	LOCAL CONST Robtarget Tr_meulage_motif_1_P373 :=[[-210.10528125,-32.02706640625,-17.9608046875],[0.732123189175605,-0.57971865199821,0.222030212103854,-0.280400615744397],[0,0,0,0],[8.999999E+09,8.999999E+09,8.999999E+09,8.999999E+09,8.999999E+09,8.999999E+09]];
	LOCAL CONST Robtarget Tr_meulage_motif_1_P374 :=[[-209.3355625,-32.6537734375,-18.0711484375],[0.732123189175605,-0.57971865199821,0.222030212103854,-0.280400615744397],[0,0,0,0],[8.999999E+09,8.999999E+09,8.999999E+09,8.999999E+09,8.999999E+09,8.999999E+09]];
	LOCAL CONST Robtarget Tr_meulage_motif_1_P375 :=[[-208.563984375,-33.28990625,-18.07105078125],[0.732123189175605,-0.57971865199821,0.222030212103854,-0.280400615744397],[0,0,0,0],[8.999999E+09,8.999999E+09,8.999999E+09,8.999999E+09,8.999999E+09,8.999999E+09]];
	LOCAL CONST Robtarget Tr_meulage_motif_1_P376 :=[[-207.79240625,-33.9260390625,-18.070953125],[0.732123189175605,-0.57971865199821,0.222030212103854,-0.280400615744397],[0,0,0,0],[8.999999E+09,8.999999E+09,8.999999E+09,8.999999E+09,8.999999E+09,8.999999E+09]];
	LOCAL CONST Robtarget Tr_meulage_motif_1_P377 :=[[-207.020828125,-34.56217578125,-18.070853515625],[0.732123189175605,-0.57971865199821,0.222030212103854,-0.280400615744397],[0,0,0,0],[8.999999E+09,8.999999E+09,8.999999E+09,8.999999E+09,8.999999E+09,8.999999E+09]];
	LOCAL CONST Robtarget Tr_meulage_motif_1_P378 :=[[-206.24925,-35.19830859375,-18.070755859375],[0.732123189175605,-0.57971865199821,0.222030212103854,-0.280400615744397],[0,0,0,0],[8.999999E+09,8.999999E+09,8.999999E+09,8.999999E+09,8.999999E+09,8.999999E+09]];
	LOCAL CONST Robtarget Tr_meulage_motif_1_P379 :=[[-205.47765625,-35.83444140625,-18.07065625],[0.732123189175605,-0.57971865199821,0.222030212103854,-0.280400615744397],[0,0,0,0],[8.999999E+09,8.999999E+09,8.999999E+09,8.999999E+09,8.999999E+09,8.999999E+09]];
	LOCAL CONST Robtarget Tr_meulage_motif_1_P380 :=[[-204.706078125,-36.47057421875,-18.07055859375],[0.732123189175605,-0.57971865199821,0.222030212103854,-0.280400615744397],[0,0,0,0],[8.999999E+09,8.999999E+09,8.999999E+09,8.999999E+09,8.999999E+09,8.999999E+09]];
	LOCAL CONST Robtarget Tr_meulage_motif_1_P381 :=[[-203.9345,-37.10670703125,-18.0704609375],[0.732123189175605,-0.57971865199821,0.222030212103854,-0.280400615744397],[0,0,0,0],[8.999999E+09,8.999999E+09,8.999999E+09,8.999999E+09,8.999999E+09,8.999999E+09]];
	LOCAL CONST Robtarget Tr_meulage_motif_1_P382 :=[[-203.162921875,-37.74283984375,-18.070361328125],[0.732123189175605,-0.57971865199821,0.222030212103854,-0.280400615744397],[0,0,0,0],[8.999999E+09,8.999999E+09,8.999999E+09,8.999999E+09,8.999999E+09,8.999999E+09]];
	LOCAL CONST Robtarget Tr_meulage_motif_1_P383 :=[[-202.39134375,-38.37897265625,-18.070263671875],[0.732123189175605,-0.57971865199821,0.222030212103854,-0.280400615744397],[0,0,0,0],[8.999999E+09,8.999999E+09,8.999999E+09,8.999999E+09,8.999999E+09,8.999999E+09]];
	LOCAL CONST Robtarget Tr_meulage_motif_1_P384 :=[[-201.619765625,-39.01510546875,-18.0701640625],[0.732123189175605,-0.57971865199821,0.222030212103854,-0.280400615744397],[0,0,0,0],[8.999999E+09,8.999999E+09,8.999999E+09,8.999999E+09,8.999999E+09,8.999999E+09]];
	LOCAL CONST Robtarget Tr_meulage_motif_1_P385 :=[[-200.8481875,-39.65123828125,-18.07006640625],[0.732123189175605,-0.57971865199821,0.222030212103854,-0.280400615744397],[0,0,0,0],[8.999999E+09,8.999999E+09,8.999999E+09,8.999999E+09,8.999999E+09,8.999999E+09]];
	LOCAL CONST Robtarget Tr_meulage_motif_1_P386 :=[[-200.076609375,-40.28737109375,-18.069966796875],[0.732123189175605,-0.57971865199821,0.222030212103854,-0.280400615744397],[0,0,0,0],[8.999999E+09,8.999999E+09,8.999999E+09,8.999999E+09,8.999999E+09,8.999999E+09]];
	LOCAL CONST Robtarget Tr_meulage_motif_1_P387 :=[[-199.30503125,-40.9235078125,-18.069869140625],[0.732123189175605,-0.57971865199821,0.222030212103854,-0.280400615744397],[0,0,0,0],[8.999999E+09,8.999999E+09,8.999999E+09,8.999999E+09,8.999999E+09,8.999999E+09]];
	LOCAL CONST Robtarget Tr_meulage_motif_1_P388 :=[[-198.533453125,-41.559640625,-18.069771484375],[0.732123189175605,-0.57971865199821,0.222030212103854,-0.280400615744397],[0,0,0,0],[8.999999E+09,8.999999E+09,8.999999E+09,8.999999E+09,8.999999E+09,8.999999E+09]];
	LOCAL CONST Robtarget Tr_meulage_motif_1_P389 :=[[-197.761875,-42.1957734375,-18.069671875],[0.732123189175605,-0.57971865199821,0.222030212103854,-0.280400615744397],[0,0,0,0],[8.999999E+09,8.999999E+09,8.999999E+09,8.999999E+09,8.999999E+09,8.999999E+09]];
	LOCAL CONST Robtarget Tr_meulage_motif_1_P390 :=[[-196.990296875,-42.83190625,-18.06957421875],[0.732123189175605,-0.57971865199821,0.222030212103854,-0.280400615744397],[0,0,0,0],[8.999999E+09,8.999999E+09,8.999999E+09,8.999999E+09,8.999999E+09,8.999999E+09]];
	LOCAL CONST Robtarget Tr_meulage_motif_1_P391 :=[[-196.21871875,-43.4680390625,-18.069474609375],[0.732123189175605,-0.57971865199821,0.222030212103854,-0.280400615744397],[0,0,0,0],[8.999999E+09,8.999999E+09,8.999999E+09,8.999999E+09,8.999999E+09,8.999999E+09]];
	LOCAL CONST Robtarget Tr_meulage_motif_1_P392 :=[[-195.447140625,-44.104171875,-18.069376953125],[0.732123189175605,-0.57971865199821,0.222030212103854,-0.280400615744397],[0,0,0,0],[8.999999E+09,8.999999E+09,8.999999E+09,8.999999E+09,8.999999E+09,8.999999E+09]];
	LOCAL CONST Robtarget Tr_meulage_motif_1_P393 :=[[-194.675546875,-44.7403046875,-18.069279296875],[0.732123189175605,-0.57971865199821,0.222030212103854,-0.280400615744397],[0,0,0,0],[8.999999E+09,8.999999E+09,8.999999E+09,8.999999E+09,8.999999E+09,8.999999E+09]];
	LOCAL CONST Robtarget Tr_meulage_motif_1_P394 :=[[-193.90396875,-45.3764375,-18.0691796875],[0.732123189175605,-0.57971865199821,0.222030212103854,-0.280400615744397],[0,0,0,0],[8.999999E+09,8.999999E+09,8.999999E+09,8.999999E+09,8.999999E+09,8.999999E+09]];
	LOCAL CONST Robtarget Tr_meulage_motif_1_P395 :=[[-193.132390625,-46.0125703125,-18.06908203125],[0.732123189175605,-0.57971865199821,0.222030212103854,-0.280400615744397],[0,0,0,0],[8.999999E+09,8.999999E+09,8.999999E+09,8.999999E+09,8.999999E+09,8.999999E+09]];
	LOCAL CONST Robtarget Tr_meulage_motif_1_P396 :=[[-192.3608125,-46.64870703125,-18.068982421875],[0.732123189175605,-0.57971865199821,0.222030212103854,-0.280400615744397],[0,0,0,0],[8.999999E+09,8.999999E+09,8.999999E+09,8.999999E+09,8.999999E+09,8.999999E+09]];
	LOCAL CONST Robtarget Tr_meulage_motif_1_P397 :=[[-191.589234375,-47.28483984375,-18.068884765625],[0.732123189175605,-0.57971865199821,0.222030212103854,-0.280400615744397],[0,0,0,0],[8.999999E+09,8.999999E+09,8.999999E+09,8.999999E+09,8.999999E+09,8.999999E+09]];
	LOCAL CONST Robtarget Tr_meulage_motif_1_P398 :=[[-190.81765625,-47.92097265625,-18.06878515625],[0.732123189175605,-0.57971865199821,0.222030212103854,-0.280400615744397],[0,0,0,0],[8.999999E+09,8.999999E+09,8.999999E+09,8.999999E+09,8.999999E+09,8.999999E+09]];
	LOCAL CONST Robtarget Tr_meulage_motif_1_P399 :=[[-190.046078125,-48.55710546875,-18.0686875],[0.732123189175605,-0.57971865199821,0.222030212103854,-0.280400615744397],[0,0,0,0],[8.999999E+09,8.999999E+09,8.999999E+09,8.999999E+09,8.999999E+09,8.999999E+09]];
	LOCAL CONST Robtarget Tr_meulage_motif_1_P400 :=[[-189.2745,-49.19323828125,-18.06858984375],[0.732123189175605,-0.57971865199821,0.222030212103854,-0.280400615744397],[0,0,0,0],[8.999999E+09,8.999999E+09,8.999999E+09,8.999999E+09,8.999999E+09,8.999999E+09]];
	LOCAL CONST Robtarget Tr_meulage_motif_1_P401 :=[[-188.502921875,-49.82937109375,-18.068490234375],[0.732123189175605,-0.57971865199821,0.222030212103854,-0.280400615744397],[0,0,0,0],[8.999999E+09,8.999999E+09,8.999999E+09,8.999999E+09,8.999999E+09,8.999999E+09]];
	LOCAL CONST Robtarget Tr_meulage_motif_1_P402 :=[[-187.73134375,-50.46550390625,-18.068392578125],[0.732123189175605,-0.57971865199821,0.222030212103854,-0.280400615744397],[0,0,0,0],[8.999999E+09,8.999999E+09,8.999999E+09,8.999999E+09,8.999999E+09,8.999999E+09]];
	LOCAL CONST Robtarget Tr_meulage_motif_1_P403 :=[[-186.959765625,-51.10163671875,-18.06829296875],[0.732123189175605,-0.57971865199821,0.222030212103854,-0.280400615744397],[0,0,0,0],[8.999999E+09,8.999999E+09,8.999999E+09,8.999999E+09,8.999999E+09,8.999999E+09]];
	LOCAL CONST Robtarget Tr_meulage_motif_1_P404 :=[[-186.1881875,-51.73776953125,-18.0681953125],[0.732123189175605,-0.57971865199821,0.222030212103854,-0.280400615744397],[0,0,0,0],[8.999999E+09,8.999999E+09,8.999999E+09,8.999999E+09,8.999999E+09,8.999999E+09]];
	LOCAL CONST Robtarget Tr_meulage_motif_1_P405 :=[[-185.416609375,-52.37390234375,-18.06809765625],[0.732123189175605,-0.57971865199821,0.222030212103854,-0.280400615744397],[0,0,0,0],[8.999999E+09,8.999999E+09,8.999999E+09,8.999999E+09,8.999999E+09,8.999999E+09]];
	LOCAL CONST Robtarget Tr_meulage_motif_1_P406 :=[[-184.64503125,-53.0100390625,-18.067998046875],[0.732123189175605,-0.57971865199821,0.222030212103854,-0.280400615744397],[0,0,0,0],[8.999999E+09,8.999999E+09,8.999999E+09,8.999999E+09,8.999999E+09,8.999999E+09]];
	LOCAL CONST Robtarget Tr_meulage_motif_1_P407 :=[[-183.8734375,-53.646171875,-18.067900390625],[0.732123189175605,-0.57971865199821,0.222030212103854,-0.280400615744397],[0,0,0,0],[8.999999E+09,8.999999E+09,8.999999E+09,8.999999E+09,8.999999E+09,8.999999E+09]];
	LOCAL CONST Robtarget Tr_meulage_motif_1_P408 :=[[-183.101859375,-54.2823046875,-18.06780078125],[0.732123189175605,-0.57971865199821,0.222030212103854,-0.280400615744397],[0,0,0,0],[8.999999E+09,8.999999E+09,8.999999E+09,8.999999E+09,8.999999E+09,8.999999E+09]];
	LOCAL CONST Robtarget Tr_meulage_motif_1_P409 :=[[-182.33028125,-54.9184375,-18.067703125],[0.732123189175605,-0.57971865199821,0.222030212103854,-0.280400615744397],[0,0,0,0],[8.999999E+09,8.999999E+09,8.999999E+09,8.999999E+09,8.999999E+09,8.999999E+09]];
	LOCAL CONST Robtarget Tr_meulage_motif_1_P410 :=[[-181.558703125,-55.5545703125,-18.067603515625],[0.732123189175605,-0.57971865199821,0.222030212103854,-0.280400615744397],[0,0,0,0],[8.999999E+09,8.999999E+09,8.999999E+09,8.999999E+09,8.999999E+09,8.999999E+09]];
	LOCAL CONST Robtarget Tr_meulage_motif_1_P411 :=[[-180.787125,-56.190703125,-18.067505859375],[0.732123189175605,-0.57971865199821,0.222030212103854,-0.280400615744397],[0,0,0,0],[8.999999E+09,8.999999E+09,8.999999E+09,8.999999E+09,8.999999E+09,8.999999E+09]];
	LOCAL CONST Robtarget Tr_meulage_motif_1_P412 :=[[-180.015546875,-56.8268359375,-18.067408203125],[0.732123189175605,-0.57971865199821,0.222030212103854,-0.280400615744397],[0,0,0,0],[8.999999E+09,8.999999E+09,8.999999E+09,8.999999E+09,8.999999E+09,8.999999E+09]];
	LOCAL CONST Robtarget Tr_meulage_motif_1_P413 :=[[-179.24396875,-57.46296875,-18.06730859375],[0.732123189175605,-0.57971865199821,0.222030212103854,-0.280400615744397],[0,0,0,0],[8.999999E+09,8.999999E+09,8.999999E+09,8.999999E+09,8.999999E+09,8.999999E+09]];
	LOCAL CONST Robtarget Tr_meulage_motif_1_P414 :=[[-178.472390625,-58.0991015625,-18.0672109375],[0.732123189175605,-0.57971865199821,0.222030212103854,-0.280400615744397],[0,0,0,0],[8.999999E+09,8.999999E+09,8.999999E+09,8.999999E+09,8.999999E+09,8.999999E+09]];
	LOCAL CONST Robtarget Tr_meulage_motif_1_P415 :=[[-177.7008125,-58.73523828125,-18.067111328125],[0.732123189175605,-0.57971865199821,0.222030212103854,-0.280400615744397],[0,0,0,0],[8.999999E+09,8.999999E+09,8.999999E+09,8.999999E+09,8.999999E+09,8.999999E+09]];
	LOCAL CONST Robtarget Tr_meulage_motif_1_P416 :=[[-176.929234375,-59.37137109375,-18.067013671875],[0.732123189175605,-0.57971865199821,0.222030212103854,-0.280400615744397],[0,0,0,0],[8.999999E+09,8.999999E+09,8.999999E+09,8.999999E+09,8.999999E+09,8.999999E+09]];
	LOCAL CONST Robtarget Tr_meulage_motif_1_P417 :=[[-176.15765625,-60.00750390625,-18.066916015625],[0.732123189175605,-0.57971865199821,0.222030212103854,-0.280400615744397],[0,0,0,0],[8.999999E+09,8.999999E+09,8.999999E+09,8.999999E+09,8.999999E+09,8.999999E+09]];
	LOCAL CONST Robtarget Tr_meulage_motif_1_P418 :=[[-175.386078125,-60.64363671875,-18.06681640625],[0.732123189175605,-0.57971865199821,0.222030212103854,-0.280400615744397],[0,0,0,0],[8.999999E+09,8.999999E+09,8.999999E+09,8.999999E+09,8.999999E+09,8.999999E+09]];
	LOCAL CONST Robtarget Tr_meulage_motif_1_P419 :=[[-174.6145,-61.27976953125,-18.06671875],[0.732123189175605,-0.57971865199821,0.222030212103854,-0.280400615744397],[0,0,0,0],[8.999999E+09,8.999999E+09,8.999999E+09,8.999999E+09,8.999999E+09,8.999999E+09]];
	LOCAL CONST Robtarget Tr_meulage_motif_1_P420 :=[[-173.842921875,-61.91590234375,-18.066619140625],[0.732123189175605,-0.57971865199821,0.222030212103854,-0.280400615744397],[0,0,0,0],[8.999999E+09,8.999999E+09,8.999999E+09,8.999999E+09,8.999999E+09,8.999999E+09]];
	LOCAL CONST Robtarget Tr_meulage_motif_1_P421 :=[[-173.071328125,-62.55203515625,-18.066521484375],[0.732123189175605,-0.57971865199821,0.222030212103854,-0.280400615744397],[0,0,0,0],[8.999999E+09,8.999999E+09,8.999999E+09,8.999999E+09,8.999999E+09,8.999999E+09]];
	LOCAL CONST Robtarget Tr_meulage_motif_1_P422 :=[[-172.29975,-63.18816796875,-18.066421875],[0.732123189175605,-0.57971865199821,0.222030212103854,-0.280400615744397],[0,0,0,0],[8.999999E+09,8.999999E+09,8.999999E+09,8.999999E+09,8.999999E+09,8.999999E+09]];
	LOCAL CONST Robtarget Tr_meulage_motif_1_P423 :=[[-171.53003125,-63.81487890625,-18.176765625],[0.732123189175605,-0.57971865199821,0.222030212103854,-0.280400615744397],[0,0,0,0],[8.999999E+09,8.999999E+09,8.999999E+09,8.999999E+09,8.999999E+09,8.999999E+09]];
	LOCAL CONST Robtarget Tr_meulage_motif_1_P424 :=[[-170.768859375,-64.43467578125,-18.285052734375],[0.732123189175605,-0.57971865199821,0.222030212103854,-0.280400615744397],[0,0,0,0],[8.999999E+09,8.999999E+09,8.999999E+09,8.999999E+09,8.999999E+09,8.999999E+09]];
	LOCAL CONST Robtarget Tr_meulage_motif_1_P425 :=[[-170.00928125,-65.05401953125,-18.38152734375],[0.732123189175605,-0.57971865199821,0.222030212103854,-0.280400615744397],[0,0,0,0],[8.999999E+09,8.999999E+09,8.999999E+09,8.999999E+09,8.999999E+09,8.999999E+09]];
	LOCAL CONST Robtarget Tr_meulage_motif_1_P426 :=[[-169.261109375,-65.66109375,-18.518021484375],[0.732123189175605,-0.57971865199821,0.222030212103854,-0.280400615744397],[0,0,0,0],[8.999999E+09,8.999999E+09,8.999999E+09,8.999999E+09,8.999999E+09,8.999999E+09]];
	LOCAL CONST Robtarget Tr_meulage_motif_1_P427 :=[[-168.36321875,-66.38365625,-18.76540625],[0.732123189175605,-0.57971865199821,0.222030212103854,-0.280400615744397],[0,0,0,0],[8.999999E+09,8.999999E+09,8.999999E+09,8.999999E+09,8.999999E+09,8.999999E+09]];
	LOCAL CONST Robtarget Tr_meulage_motif_1_P428 :=[[-167.63828125,-66.9588515625,-19.079759765625],[0.732123189175605,-0.57971865199821,0.222030212103854,-0.280400615744397],[0,0,0,0],[8.999999E+09,8.999999E+09,8.999999E+09,8.999999E+09,8.999999E+09,8.999999E+09]];
	LOCAL CONST Robtarget Tr_meulage_motif_1_degg1 :=[[-174.140419929152,-74.2022127652547,-21.3723371543949],[0.732123189175605,-0.57971865199821,0.222030212103854,-0.280400615744397],[0,0,0,0],[8.999999E+09,8.999999E+09,8.999999E+09,8.999999E+09,8.999999E+09,8.999999E+09]];
	LOCAL CONST Robtarget Tr_meulage_motif_1_degg2 :=[[-297.681054833048,-211.826075617593,-64.9313075410234],[0.732123189175605,-0.57971865199821,0.222030212103854,-0.280400615744397],[0,0,0,0],[8.999999E+09,8.999999E+09,8.999999E+09,8.999999E+09,8.999999E+09,8.999999E+09]];
	LOCAL CONST Robtarget Tr_meulage_motif_2_App1 :=[[84.4850303618467,-122.237799931102,-198.639888227745],[-7.71783197556249E-06,0.00508283936343101,0.0015183882137476,0.999985929491847],[0,0,0,0],[8.999999E+09,8.999999E+09,8.999999E+09,8.999999E+09,8.999999E+09,8.999999E+09]];
	LOCAL CONST Robtarget Tr_meulage_motif_2_App2 :=[[86.4164776899673,-121.660805621555,-8.65058171607476],[-7.71783197556249E-06,0.00508283936343101,0.0015183882137476,0.999985929491847],[0,0,0,0],[8.999999E+09,8.999999E+09,8.999999E+09,8.999999E+09,8.999999E+09,8.999999E+09]];
	LOCAL CONST Robtarget Tr_meulage_motif_2_P0 :=[[86.5181328125,-121.6304375,1.34885546875],[-7.71783197556249E-06,0.00508283936343101,0.0015183882137476,0.999985929491847],[0,0,0,0],[8.999999E+09,8.999999E+09,8.999999E+09,8.999999E+09,8.999999E+09,8.999999E+09]];
	LOCAL CONST Robtarget Tr_meulage_motif_2_P1 :=[[87.442578125,-121.2491953125,1.34139868164062],[-7.71783197556249E-06,0.00508283936343101,0.0015183882137476,0.999985929491847],[0,0,0,0],[8.999999E+09,8.999999E+09,8.999999E+09,8.999999E+09,8.999999E+09,8.999999E+09]];
	LOCAL CONST Robtarget Tr_meulage_motif_2_P2 :=[[88.3670234375,-120.8679609375,1.33394177246094],[-7.71783197556249E-06,0.00508283936343101,0.0015183882137476,0.999985929491847],[0,0,0,0],[8.999999E+09,8.999999E+09,8.999999E+09,8.999999E+09,8.999999E+09,8.999999E+09]];
	LOCAL CONST Robtarget Tr_meulage_motif_2_P3 :=[[89.29146875,-120.48671875,1.32648486328125],[-7.71783197556249E-06,0.00508283936343101,0.0015183882137476,0.999985929491847],[0,0,0,0],[8.999999E+09,8.999999E+09,8.999999E+09,8.999999E+09,8.999999E+09,8.999999E+09]];
	LOCAL CONST Robtarget Tr_meulage_motif_2_P4 :=[[90.2159140625,-120.1054765625,1.31902795410156],[-7.71783197556249E-06,0.00508283936343101,0.0015183882137476,0.999985929491847],[0,0,0,0],[8.999999E+09,8.999999E+09,8.999999E+09,8.999999E+09,8.999999E+09,8.999999E+09]];
	LOCAL CONST Robtarget Tr_meulage_motif_2_P5 :=[[91.140359375,-119.7242421875,1.31157116699219],[-7.71783197556249E-06,0.00508283936343101,0.0015183882137476,0.999985929491847],[0,0,0,0],[8.999999E+09,8.999999E+09,8.999999E+09,8.999999E+09,8.999999E+09,8.999999E+09]];
	LOCAL CONST Robtarget Tr_meulage_motif_2_P6 :=[[92.0648046875,-119.343,1.3041142578125],[-7.71783197556249E-06,0.00508283936343101,0.0015183882137476,0.999985929491847],[0,0,0,0],[8.999999E+09,8.999999E+09,8.999999E+09,8.999999E+09,8.999999E+09,8.999999E+09]];
	LOCAL CONST Robtarget Tr_meulage_motif_2_P7 :=[[92.98925,-118.9617578125,1.29665734863281],[-7.71783197556249E-06,0.00508283936343101,0.0015183882137476,0.999985929491847],[0,0,0,0],[8.999999E+09,8.999999E+09,8.999999E+09,8.999999E+09,8.999999E+09,8.999999E+09]];
	LOCAL CONST Robtarget Tr_meulage_motif_2_P8 :=[[93.913703125,-118.5805234375,1.28920043945313],[-7.71783197556249E-06,0.00508283936343101,0.0015183882137476,0.999985929491847],[0,0,0,0],[8.999999E+09,8.999999E+09,8.999999E+09,8.999999E+09,8.999999E+09,8.999999E+09]];
	LOCAL CONST Robtarget Tr_meulage_motif_2_P9 :=[[94.8381484375,-118.19928125,1.28174365234375],[-7.71783197556249E-06,0.00508283936343101,0.0015183882137476,0.999985929491847],[0,0,0,0],[8.999999E+09,8.999999E+09,8.999999E+09,8.999999E+09,8.999999E+09,8.999999E+09]];
	LOCAL CONST Robtarget Tr_meulage_motif_2_P10 :=[[95.76259375,-117.8180390625,1.27428674316406],[-7.71783197556249E-06,0.00508283936343101,0.0015183882137476,0.999985929491847],[0,0,0,0],[8.999999E+09,8.999999E+09,8.999999E+09,8.999999E+09,8.999999E+09,8.999999E+09]];
	LOCAL CONST Robtarget Tr_meulage_motif_2_P11 :=[[96.6870390625,-117.4368046875,1.26682983398438],[-7.71783197556249E-06,0.00508283936343101,0.0015183882137476,0.999985929491847],[0,0,0,0],[8.999999E+09,8.999999E+09,8.999999E+09,8.999999E+09,8.999999E+09,8.999999E+09]];
	LOCAL CONST Robtarget Tr_meulage_motif_2_P12 :=[[97.611484375,-117.0555625,1.25937292480469],[-7.71783197556249E-06,0.00508283936343101,0.0015183882137476,0.999985929491847],[0,0,0,0],[8.999999E+09,8.999999E+09,8.999999E+09,8.999999E+09,8.999999E+09,8.999999E+09]];
	LOCAL CONST Robtarget Tr_meulage_motif_2_P13 :=[[98.5359296875,-116.6743203125,1.25191613769531],[-7.71783197556249E-06,0.00508283936343101,0.0015183882137476,0.999985929491847],[0,0,0,0],[8.999999E+09,8.999999E+09,8.999999E+09,8.999999E+09,8.999999E+09,8.999999E+09]];
	LOCAL CONST Robtarget Tr_meulage_motif_2_P14 :=[[99.460375,-116.293078125,1.24445922851563],[-7.71783197556249E-06,0.00508283936343101,0.0015183882137476,0.999985929491847],[0,0,0,0],[8.999999E+09,8.999999E+09,8.999999E+09,8.999999E+09,8.999999E+09,8.999999E+09]];
	LOCAL CONST Robtarget Tr_meulage_motif_2_P15 :=[[100.3848203125,-115.91184375,1.23700231933594],[-7.71783197556249E-06,0.00508283936343101,0.0015183882137476,0.999985929491847],[0,0,0,0],[8.999999E+09,8.999999E+09,8.999999E+09,8.999999E+09,8.999999E+09,8.999999E+09]];
	LOCAL CONST Robtarget Tr_meulage_motif_2_P16 :=[[101.309265625,-115.5306015625,1.22954553222656],[-7.71783197556249E-06,0.00508283936343101,0.0015183882137476,0.999985929491847],[0,0,0,0],[8.999999E+09,8.999999E+09,8.999999E+09,8.999999E+09,8.999999E+09,8.999999E+09]];
	LOCAL CONST Robtarget Tr_meulage_motif_2_P17 :=[[102.2337109375,-115.149359375,1.22208862304688],[-7.71783197556249E-06,0.00508283936343101,0.0015183882137476,0.999985929491847],[0,0,0,0],[8.999999E+09,8.999999E+09,8.999999E+09,8.999999E+09,8.999999E+09,8.999999E+09]];
	LOCAL CONST Robtarget Tr_meulage_motif_2_P18 :=[[103.1581640625,-114.768125,1.21463171386719],[-7.71783197556249E-06,0.00508283936343101,0.0015183882137476,0.999985929491847],[0,0,0,0],[8.999999E+09,8.999999E+09,8.999999E+09,8.999999E+09,8.999999E+09,8.999999E+09]];
	LOCAL CONST Robtarget Tr_meulage_motif_2_P19 :=[[104.0335625,-114.2875,1.20517932128906],[-7.71783197556249E-06,0.00508283936343101,0.0015183882137476,0.999985929491847],[0,0,0,0],[8.999999E+09,8.999999E+09,8.999999E+09,8.999999E+09,8.999999E+09,8.999999E+09]];
	LOCAL CONST Robtarget Tr_meulage_motif_2_P20 :=[[104.8280234375,-113.73146875,1.19420471191406],[-7.71783197556249E-06,0.00508283936343101,0.0015183882137476,0.999985929491847],[0,0,0,0],[8.999999E+09,8.999999E+09,8.999999E+09,8.999999E+09,8.999999E+09,8.999999E+09]];
	LOCAL CONST Robtarget Tr_meulage_motif_2_P21 :=[[105.51265625,-113.155125,1.1828046875],[-7.71783197556249E-06,0.00508283936343101,0.0015183882137476,0.999985929491847],[0,0,0,0],[8.999999E+09,8.999999E+09,8.999999E+09,8.999999E+09,8.999999E+09,8.999999E+09]];
	LOCAL CONST Robtarget Tr_meulage_motif_2_P22 :=[[106.1007109375,-112.6141796875,1.17209509277344],[-7.71783197556249E-06,0.00508283936343101,0.0015183882137476,0.999985929491847],[0,0,0,0],[8.999999E+09,8.999999E+09,8.999999E+09,8.999999E+09,8.999999E+09,8.999999E+09]];
	LOCAL CONST Robtarget Tr_meulage_motif_2_P23 :=[[106.8836484375,-111.6249453125,1.15245812988281],[-7.71783197556249E-06,0.00508283936343101,0.0015183882137476,0.999985929491847],[0,0,0,0],[8.999999E+09,8.999999E+09,8.999999E+09,8.999999E+09,8.999999E+09,8.999999E+09]];
	LOCAL CONST Robtarget Tr_meulage_motif_2_P24 :=[[107.5069453125,-110.4511484375,1.12910302734375],[-7.71783197556249E-06,0.00508283936343101,0.0015183882137476,0.999985929491847],[0,0,0,0],[8.999999E+09,8.999999E+09,8.999999E+09,8.999999E+09,8.999999E+09,8.999999E+09]];
	LOCAL CONST Robtarget Tr_meulage_motif_2_P25 :=[[107.900140625,-109.1816640625,1.10379382324219],[-7.71783197556249E-06,0.00508283936343101,0.0015183882137476,0.999985929491847],[0,0,0,0],[8.999999E+09,8.999999E+09,8.999999E+09,8.999999E+09,8.999999E+09,8.999999E+09]];
	LOCAL CONST Robtarget Tr_meulage_motif_2_P26 :=[[107.925796875,-107.9639140625,1.07945336914062],[-7.71783197556249E-06,0.00508283936343101,0.0015183882137476,0.999985929491847],[0,0,0,0],[8.999999E+09,8.999999E+09,8.999999E+09,8.999999E+09,8.999999E+09,8.999999E+09]];
	LOCAL CONST Robtarget Tr_meulage_motif_2_P27 :=[[107.6854375,-107.3103359375,1.06634436035156],[-7.71783197556249E-06,0.00508283936343101,0.0015183882137476,0.999985929491847],[0,0,0,0],[8.999999E+09,8.999999E+09,8.999999E+09,8.999999E+09,8.999999E+09,8.999999E+09]];
	LOCAL CONST Robtarget Tr_meulage_motif_2_P28 :=[[107.433296875,-106.699171875,1.05408117675781],[-7.71783197556249E-06,0.00508283936343101,0.0015183882137476,0.999985929491847],[0,0,0,0],[8.999999E+09,8.999999E+09,8.999999E+09,8.999999E+09,8.999999E+09,8.999999E+09]];
	LOCAL CONST Robtarget Tr_meulage_motif_2_P29 :=[[107.130484375,-106.1090703125,1.04222998046875],[-7.71783197556249E-06,0.00508283936343101,0.0015183882137476,0.999985929491847],[0,0,0,0],[8.999999E+09,8.999999E+09,8.999999E+09,8.999999E+09,8.999999E+09,8.999999E+09]];
	LOCAL CONST Robtarget Tr_meulage_motif_2_P30 :=[[106.249796875,-105.2807109375,1.02551257324219],[-7.71783197556249E-06,0.00508283936343101,0.0015183882137476,0.999985929491847],[0,0,0,0],[8.999999E+09,8.999999E+09,8.999999E+09,8.999999E+09,8.999999E+09,8.999999E+09]];
	LOCAL CONST Robtarget Tr_meulage_motif_2_P31 :=[[105.074046875,-104.67690625,1.01323187255859],[-7.71783197556249E-06,0.00508283936343101,0.0015183882137476,0.999985929491847],[0,0,0,0],[8.999999E+09,8.999999E+09,8.999999E+09,8.999999E+09,8.999999E+09,8.999999E+09]];
	LOCAL CONST Robtarget Tr_meulage_motif_2_P32 :=[[103.81190625,-104.30096875,1.00549133300781],[-7.71783197556249E-06,0.00508283936343101,0.0015183882137476,0.999985929491847],[0,0,0,0],[8.999999E+09,8.999999E+09,8.999999E+09,8.999999E+09,8.999999E+09,8.999999E+09]];
	LOCAL CONST Robtarget Tr_meulage_motif_2_P33 :=[[103.0258203125,-104.197140625,1.00327545166016],[-7.71783197556249E-06,0.00508283936343101,0.0015183882137476,0.999985929491847],[0,0,0,0],[8.999999E+09,8.999999E+09,8.999999E+09,8.999999E+09,8.999999E+09,8.999999E+09]];
	LOCAL CONST Robtarget Tr_meulage_motif_2_P34 :=[[101.769265625,-104.1880703125,1.00287017822266],[-7.71783197556249E-06,0.00508283936343101,0.0015183882137476,0.999985929491847],[0,0,0,0],[8.999999E+09,8.999999E+09,8.999999E+09,8.999999E+09,8.999999E+09,8.999999E+09]];
	LOCAL CONST Robtarget Tr_meulage_motif_2_P35 :=[[100.887375,-104.266140625,1.00427368164063],[-7.71783197556249E-06,0.00508283936343101,0.0015183882137476,0.999985929491847],[0,0,0,0],[8.999999E+09,8.999999E+09,8.999999E+09,8.999999E+09,8.999999E+09,8.999999E+09]];
	LOCAL CONST Robtarget Tr_meulage_motif_2_P36 :=[[99.947828125,-104.4324765625,1.00743151855469],[-7.71783197556249E-06,0.00508283936343101,0.0015183882137476,0.999985929491847],[0,0,0,0],[8.999999E+09,8.999999E+09,8.999999E+09,8.999999E+09,8.999999E+09,8.999999E+09]];
	LOCAL CONST Robtarget Tr_meulage_motif_2_P37 :=[[98.999015625,-104.7063125,1.01273693847656],[-7.71783197556249E-06,0.00508283936343101,0.0015183882137476,0.999985929491847],[0,0,0,0],[8.999999E+09,8.999999E+09,8.999999E+09,8.999999E+09,8.999999E+09,8.999999E+09]];
	LOCAL CONST Robtarget Tr_meulage_motif_2_P38 :=[[98.0392734375,-104.9825,1.01808734130859],[-7.71783197556249E-06,0.00508283936343101,0.0015183882137476,0.999985929491847],[0,0,0,0],[8.999999E+09,8.999999E+09,8.999999E+09,8.999999E+09,8.999999E+09,8.999999E+09]];
	LOCAL CONST Robtarget Tr_meulage_motif_2_P39 :=[[97.114828125,-105.3637421875,1.02554418945312],[-7.71783197556249E-06,0.00508283936343101,0.0015183882137476,0.999985929491847],[0,0,0,0],[8.999999E+09,8.999999E+09,8.999999E+09,8.999999E+09,8.999999E+09,8.999999E+09]];
	LOCAL CONST Robtarget Tr_meulage_motif_2_P40 :=[[96.1903828125,-105.744984375,1.03300109863281],[-7.71783197556249E-06,0.00508283936343101,0.0015183882137476,0.999985929491847],[0,0,0,0],[8.999999E+09,8.999999E+09,8.999999E+09,8.999999E+09,8.999999E+09,8.999999E+09]];
	LOCAL CONST Robtarget Tr_meulage_motif_2_P41 :=[[95.2659375,-106.12621875,1.0404580078125],[-7.71783197556249E-06,0.00508283936343101,0.0015183882137476,0.999985929491847],[0,0,0,0],[8.999999E+09,8.999999E+09,8.999999E+09,8.999999E+09,8.999999E+09,8.999999E+09]];
	LOCAL CONST Robtarget Tr_meulage_motif_2_P42 :=[[94.3414921875,-106.5074609375,1.04791491699219],[-7.71783197556249E-06,0.00508283936343101,0.0015183882137476,0.999985929491847],[0,0,0,0],[8.999999E+09,8.999999E+09,8.999999E+09,8.999999E+09,8.999999E+09,8.999999E+09]];
	LOCAL CONST Robtarget Tr_meulage_motif_2_P43 :=[[93.417046875,-106.888703125,1.05537170410156],[-7.71783197556249E-06,0.00508283936343101,0.0015183882137476,0.999985929491847],[0,0,0,0],[8.999999E+09,8.999999E+09,8.999999E+09,8.999999E+09,8.999999E+09,8.999999E+09]];
	LOCAL CONST Robtarget Tr_meulage_motif_2_P44 :=[[92.4926015625,-107.2699375,1.06282861328125],[-7.71783197556249E-06,0.00508283936343101,0.0015183882137476,0.999985929491847],[0,0,0,0],[8.999999E+09,8.999999E+09,8.999999E+09,8.999999E+09,8.999999E+09,8.999999E+09]];
	LOCAL CONST Robtarget Tr_meulage_motif_2_P45 :=[[91.56815625,-107.6511796875,1.07028552246094],[-7.71783197556249E-06,0.00508283936343101,0.0015183882137476,0.999985929491847],[0,0,0,0],[8.999999E+09,8.999999E+09,8.999999E+09,8.999999E+09,8.999999E+09,8.999999E+09]];
	LOCAL CONST Robtarget Tr_meulage_motif_2_P46 :=[[90.643703125,-108.032421875,1.07774243164062],[-7.71783197556249E-06,0.00508283936343101,0.0015183882137476,0.999985929491847],[0,0,0,0],[8.999999E+09,8.999999E+09,8.999999E+09,8.999999E+09,8.999999E+09,8.999999E+09]];
	LOCAL CONST Robtarget Tr_meulage_motif_2_P47 :=[[89.7192578125,-108.41365625,1.08519921875],[-7.71783197556249E-06,0.00508283936343101,0.0015183882137476,0.999985929491847],[0,0,0,0],[8.999999E+09,8.999999E+09,8.999999E+09,8.999999E+09,8.999999E+09,8.999999E+09]];
	LOCAL CONST Robtarget Tr_meulage_motif_2_P48 :=[[88.7948125,-108.7948984375,1.09265612792969],[-7.71783197556249E-06,0.00508283936343101,0.0015183882137476,0.999985929491847],[0,0,0,0],[8.999999E+09,8.999999E+09,8.999999E+09,8.999999E+09,8.999999E+09,8.999999E+09]];
	LOCAL CONST Robtarget Tr_meulage_motif_2_P49 :=[[87.8350703125,-109.0710859375,1.09800646972656],[-7.71783197556249E-06,0.00508283936343101,0.0015183882137476,0.999985929491847],[0,0,0,0],[8.999999E+09,8.999999E+09,8.999999E+09,8.999999E+09,8.999999E+09,8.999999E+09]];
	LOCAL CONST Robtarget Tr_meulage_motif_2_P50 :=[[86.8795546875,-109.236734375,1.10114782714844],[-7.71783197556249E-06,0.00508283936343101,0.0015183882137476,0.999985929491847],[0,0,0,0],[8.999999E+09,8.999999E+09,8.999999E+09,8.999999E+09,8.999999E+09,8.999999E+09]];
	LOCAL CONST Robtarget Tr_meulage_motif_2_P51 :=[[85.987609375,-109.3105703125,1.10246496582031],[-7.71783197556249E-06,0.00508283936343101,0.0015183882137476,0.999985929491847],[0,0,0,0],[8.999999E+09,8.999999E+09,8.999999E+09,8.999999E+09,8.999999E+09,8.999999E+09]];
	LOCAL CONST Robtarget Tr_meulage_motif_2_P52 :=[[85.2138828125,-109.300703125,1.10212976074219],[-7.71783197556249E-06,0.00508283936343101,0.0015183882137476,0.999985929491847],[0,0,0,0],[8.999999E+09,8.999999E+09,8.999999E+09,8.999999E+09,8.999999E+09,8.999999E+09]];
	LOCAL CONST Robtarget Tr_meulage_motif_2_P53 :=[[84.0049453125,-109.082734375,1.097556640625],[-7.71783197556249E-06,0.00508283936343101,0.0015183882137476,0.999985929491847],[0,0,0,0],[8.999999E+09,8.999999E+09,8.999999E+09,8.999999E+09,8.999999E+09,8.999999E+09]];
	LOCAL CONST Robtarget Tr_meulage_motif_2_P54 :=[[82.8272265625,-108.5929609375,1.08755541992188],[-7.71783197556249E-06,0.00508283936343101,0.0015183882137476,0.999985929491847],[0,0,0,0],[8.999999E+09,8.999999E+09,8.999999E+09,8.999999E+09,8.999999E+09,8.999999E+09]];
	LOCAL CONST Robtarget Tr_meulage_motif_2_P55 :=[[81.9338125,-107.830109375,1.07214538574219],[-7.71783197556249E-06,0.00508283936343101,0.0015183882137476,0.999985929491847],[0,0,0,0],[8.999999E+09,8.999999E+09,8.999999E+09,8.999999E+09,8.999999E+09,8.999999E+09]];
	LOCAL CONST Robtarget Tr_meulage_motif_2_P56 :=[[81.4986640625,-107.25984375,1.06066711425781],[-7.71783197556249E-06,0.00508283936343101,0.0015183882137476,0.999985929491847],[0,0,0,0],[8.999999E+09,8.999999E+09,8.999999E+09,8.999999E+09,8.999999E+09,8.999999E+09]];
	LOCAL CONST Robtarget Tr_meulage_motif_2_P57 :=[[81.14603125,-106.5725,1.04686303710938],[-7.71783197556249E-06,0.00508283936343101,0.0015183882137476,0.999985929491847],[0,0,0,0],[8.999999E+09,8.999999E+09,8.999999E+09,8.999999E+09,8.999999E+09,8.999999E+09]];
	LOCAL CONST Robtarget Tr_meulage_motif_2_P58 :=[[80.9143515625,-105.8354140625,1.03208618164063],[-7.71783197556249E-06,0.00508283936343101,0.0015183882137476,0.999985929491847],[0,0,0,0],[8.999999E+09,8.999999E+09,8.999999E+09,8.999999E+09,8.999999E+09,8.999999E+09]];
	LOCAL CONST Robtarget Tr_meulage_motif_2_P59 :=[[80.8796484375,-104.651140625,1.00840417480469],[-7.71783197556249E-06,0.00508283936343101,0.0015183882137476,0.999985929491847],[0,0,0,0],[8.999999E+09,8.999999E+09,8.999999E+09,8.999999E+09,8.999999E+09,8.999999E+09]];
	LOCAL CONST Robtarget Tr_meulage_motif_2_P60 :=[[81.039328125,-103.951859375,0.994452819824219],[-7.71783197556249E-06,0.00508283936343101,0.0015183882137476,0.999985929491847],[0,0,0,0],[8.999999E+09,8.999999E+09,8.999999E+09,8.999999E+09,8.999999E+09,8.999999E+09]];
	LOCAL CONST Robtarget Tr_meulage_motif_2_P61 :=[[81.52115625,-102.79371875,0.971385375976562],[-7.71783197556249E-06,0.00508283936343101,0.0015183882137476,0.999985929491847],[0,0,0,0],[8.999999E+09,8.999999E+09,8.999999E+09,8.999999E+09,8.999999E+09,8.999999E+09]];
	LOCAL CONST Robtarget Tr_meulage_motif_2_P62 :=[[81.904609375,-102.1875,0.959334289550781],[-7.71783197556249E-06,0.00508283936343101,0.0015183882137476,0.999985929491847],[0,0,0,0],[8.999999E+09,8.999999E+09,8.999999E+09,8.999999E+09,8.999999E+09,8.999999E+09]];
	LOCAL CONST Robtarget Tr_meulage_motif_2_P63 :=[[82.7305859375,-101.258421875,0.94090771484375],[-7.71783197556249E-06,0.00508283936343101,0.0015183882137476,0.999985929491847],[0,0,0,0],[8.999999E+09,8.999999E+09,8.999999E+09,8.999999E+09,8.999999E+09,8.999999E+09]];
	LOCAL CONST Robtarget Tr_meulage_motif_2_P64 :=[[83.381125,-100.6705546875,0.929271118164062],[-7.71783197556249E-06,0.00508283936343101,0.0015183882137476,0.999985929491847],[0,0,0,0],[8.999999E+09,8.999999E+09,8.999999E+09,8.999999E+09,8.999999E+09,8.999999E+09]];
	LOCAL CONST Robtarget Tr_meulage_motif_2_P65 :=[[84.1647421875,-100.1262578125,0.918529357910156],[-7.71783197556249E-06,0.00508283936343101,0.0015183882137476,0.999985929491847],[0,0,0,0],[8.999999E+09,8.999999E+09,8.999999E+09,8.999999E+09,8.999999E+09,8.999999E+09]];
	LOCAL CONST Robtarget Tr_meulage_motif_2_P66 :=[[85.030734375,-99.6516796875,0.909195983886719],[-7.71783197556249E-06,0.00508283936343101,0.0015183882137476,0.999985929491847],[0,0,0,0],[8.999999E+09,8.999999E+09,8.999999E+09,8.999999E+09,8.999999E+09,8.999999E+09]];
	LOCAL CONST Robtarget Tr_meulage_motif_2_P67 :=[[85.9061328125,-99.1710546875,0.899743591308594],[-7.71783197556249E-06,0.00508283936343101,0.0015183882137476,0.999985929491847],[0,0,0,0],[8.999999E+09,8.999999E+09,8.999999E+09,8.999999E+09,8.999999E+09,8.999999E+09]];
	LOCAL CONST Robtarget Tr_meulage_motif_2_P68 :=[[86.830578125,-98.7898203125,0.892286682128906],[-7.71783197556249E-06,0.00508283936343101,0.0015183882137476,0.999985929491847],[0,0,0,0],[8.999999E+09,8.999999E+09,8.999999E+09,8.999999E+09,8.999999E+09,8.999999E+09]];
	LOCAL CONST Robtarget Tr_meulage_motif_2_P69 :=[[87.7550234375,-98.408578125,0.884829833984375],[-7.71783197556249E-06,0.00508283936343101,0.0015183882137476,0.999985929491847],[0,0,0,0],[8.999999E+09,8.999999E+09,8.999999E+09,8.999999E+09,8.999999E+09,8.999999E+09]];
	LOCAL CONST Robtarget Tr_meulage_motif_2_P70 :=[[88.6794765625,-98.0273359375,0.877372924804688],[-7.71783197556249E-06,0.00508283936343101,0.0015183882137476,0.999985929491847],[0,0,0,0],[8.999999E+09,8.999999E+09,8.999999E+09,8.999999E+09,8.999999E+09,8.999999E+09]];
	LOCAL CONST Robtarget Tr_meulage_motif_2_P71 :=[[89.603921875,-97.6461015625,0.869916076660156],[-7.71783197556249E-06,0.00508283936343101,0.0015183882137476,0.999985929491847],[0,0,0,0],[8.999999E+09,8.999999E+09,8.999999E+09,8.999999E+09,8.999999E+09,8.999999E+09]];
	LOCAL CONST Robtarget Tr_meulage_motif_2_P72 :=[[90.5283671875,-97.264859375,0.862459167480469],[-7.71783197556249E-06,0.00508283936343101,0.0015183882137476,0.999985929491847],[0,0,0,0],[8.999999E+09,8.999999E+09,8.999999E+09,8.999999E+09,8.999999E+09,8.999999E+09]];
	LOCAL CONST Robtarget Tr_meulage_motif_2_P73 :=[[91.4528125,-96.8836171875,0.855002319335938],[-7.71783197556249E-06,0.00508283936343101,0.0015183882137476,0.999985929491847],[0,0,0,0],[8.999999E+09,8.999999E+09,8.999999E+09,8.999999E+09,8.999999E+09,8.999999E+09]];
	LOCAL CONST Robtarget Tr_meulage_motif_2_P74 :=[[92.3772578125,-96.5023828125,0.84754541015625],[-7.71783197556249E-06,0.00508283936343101,0.0015183882137476,0.999985929491847],[0,0,0,0],[8.999999E+09,8.999999E+09,8.999999E+09,8.999999E+09,8.999999E+09,8.999999E+09]];
	LOCAL CONST Robtarget Tr_meulage_motif_2_P75 :=[[93.301703125,-96.121140625,0.840088562011719],[-7.71783197556249E-06,0.00508283936343101,0.0015183882137476,0.999985929491847],[0,0,0,0],[8.999999E+09,8.999999E+09,8.999999E+09,8.999999E+09,8.999999E+09,8.999999E+09]];
	LOCAL CONST Robtarget Tr_meulage_motif_2_P76 :=[[94.2261484375,-95.7398984375,0.832631713867187],[-7.71783197556249E-06,0.00508283936343101,0.0015183882137476,0.999985929491847],[0,0,0,0],[8.999999E+09,8.999999E+09,8.999999E+09,8.999999E+09,8.999999E+09,8.999999E+09]];
	LOCAL CONST Robtarget Tr_meulage_motif_2_P77 :=[[95.15059375,-95.3586640625,0.8251748046875],[-7.71783197556249E-06,0.00508283936343101,0.0015183882137476,0.999985929491847],[0,0,0,0],[8.999999E+09,8.999999E+09,8.999999E+09,8.999999E+09,8.999999E+09,8.999999E+09]];
	LOCAL CONST Robtarget Tr_meulage_motif_2_P78 :=[[96.0259921875,-94.8780390625,0.815722351074219],[-7.71783197556249E-06,0.00508283936343101,0.0015183882137476,0.999985929491847],[0,0,0,0],[8.999999E+09,8.999999E+09,8.999999E+09,8.999999E+09,8.999999E+09,8.999999E+09]];
	LOCAL CONST Robtarget Tr_meulage_motif_2_P79 :=[[96.820453125,-94.322,0.804747863769531],[-7.71783197556249E-06,0.00508283936343101,0.0015183882137476,0.999985929491847],[0,0,0,0],[8.999999E+09,8.999999E+09,8.999999E+09,8.999999E+09,8.999999E+09,8.999999E+09]];
	LOCAL CONST Robtarget Tr_meulage_motif_2_P80 :=[[97.50509375,-93.74565625,0.793347717285156],[-7.71783197556249E-06,0.00508283936343101,0.0015183882137476,0.999985929491847],[0,0,0,0],[8.999999E+09,8.999999E+09,8.999999E+09,8.999999E+09,8.999999E+09,8.999999E+09]];
	LOCAL CONST Robtarget Tr_meulage_motif_2_P81 :=[[98.0931484375,-93.2047109375,0.782638122558594],[-7.71783197556249E-06,0.00508283936343101,0.0015183882137476,0.999985929491847],[0,0,0,0],[8.999999E+09,8.999999E+09,8.999999E+09,8.999999E+09,8.999999E+09,8.999999E+09]];
	LOCAL CONST Robtarget Tr_meulage_motif_2_P82 :=[[98.8760859375,-92.215484375,0.763001220703125],[-7.71783197556249E-06,0.00508283936343101,0.0015183882137476,0.999985929491847],[0,0,0,0],[8.999999E+09,8.999999E+09,8.999999E+09,8.999999E+09,8.999999E+09,8.999999E+09]];
	LOCAL CONST Robtarget Tr_meulage_motif_2_P83 :=[[99.419640625,-91.024484375,0.739287963867188],[-7.71783197556249E-06,0.00508283936343101,0.0015183882137476,0.999985929491847],[0,0,0,0],[8.999999E+09,8.999999E+09,8.999999E+09,8.999999E+09,8.999999E+09,8.999999E+09]];
	LOCAL CONST Robtarget Tr_meulage_motif_2_P84 :=[[99.568640625,-89.788515625,0.714605285644531],[-7.71783197556249E-06,0.00508283936343101,0.0015183882137476,0.999985929491847],[0,0,0,0],[8.999999E+09,8.999999E+09,8.999999E+09,8.999999E+09,8.999999E+09,8.999999E+09]];
	LOCAL CONST Robtarget Tr_meulage_motif_2_P85 :=[[99.3498046875,-88.8141484375,0.695086975097656],[-7.71783197556249E-06,0.00508283936343101,0.0015183882137476,0.999985929491847],[0,0,0,0],[8.999999E+09,8.999999E+09,8.999999E+09,8.999999E+09,8.999999E+09,8.999999E+09]];
	LOCAL CONST Robtarget Tr_meulage_motif_2_P86 :=[[99.1502265625,-88.6751171875,0.692271850585938],[-7.71783197556249E-06,0.00508283936343101,0.0015183882137476,0.999985929491847],[0,0,0,0],[8.999999E+09,8.999999E+09,8.999999E+09,8.999999E+09,8.999999E+09,8.999999E+09]];
	LOCAL CONST Robtarget Tr_meulage_motif_2_P87 :=[[98.7591875,-88.050765625,0.67972021484375],[-7.71783197556249E-06,0.00508283936343101,0.0015183882137476,0.999985929491847],[0,0,0,0],[8.999999E+09,8.999999E+09,8.999999E+09,8.999999E+09,8.999999E+09,8.999999E+09]];
	LOCAL CONST Robtarget Tr_meulage_motif_2_P88 :=[[97.769609375,-87.4455859375,0.667445251464844],[-7.71783197556249E-06,0.00508283936343101,0.0015183882137476,0.999985929491847],[0,0,0,0],[8.999999E+09,8.999999E+09,8.999999E+09,8.999999E+09,8.999999E+09,8.999999E+09]];
	LOCAL CONST Robtarget Tr_meulage_motif_2_P89 :=[[97.0772578125,-87.2294921875,0.663001708984375],[-7.71783197556249E-06,0.00508283936343101,0.0015183882137476,0.999985929491847],[0,0,0,0],[8.999999E+09,8.999999E+09,8.999999E+09,8.999999E+09,8.999999E+09,8.999999E+09]];
	LOCAL CONST Robtarget Tr_meulage_motif_2_P90 :=[[95.8300859375,-87.1701484375,0.661593078613281],[-7.71783197556249E-06,0.00508283936343101,0.0015183882137476,0.999985929491847],[0,0,0,0],[8.999999E+09,8.999999E+09,8.999999E+09,8.999999E+09,8.999999E+09,8.999999E+09]];
	LOCAL CONST Robtarget Tr_meulage_motif_2_P91 :=[[94.9481953125,-87.24821875,0.66299658203125],[-7.71783197556249E-06,0.00508283936343101,0.0015183882137476,0.999985929491847],[0,0,0,0],[8.999999E+09,8.999999E+09,8.999999E+09,8.999999E+09,8.999999E+09,8.999999E+09]];
	LOCAL CONST Robtarget Tr_meulage_motif_2_P92 :=[[94.0086484375,-87.4145546875,0.666154418945312],[-7.71783197556249E-06,0.00508283936343101,0.0015183882137476,0.999985929491847],[0,0,0,0],[8.999999E+09,8.999999E+09,8.999999E+09,8.999999E+09,8.999999E+09,8.999999E+09]];
	LOCAL CONST Robtarget Tr_meulage_motif_2_P93 :=[[93.0598359375,-87.688390625,0.671459899902344],[-7.71783197556249E-06,0.00508283936343101,0.0015183882137476,0.999985929491847],[0,0,0,0],[8.999999E+09,8.999999E+09,8.999999E+09,8.999999E+09,8.999999E+09,8.999999E+09]];
	LOCAL CONST Robtarget Tr_meulage_motif_2_P94 :=[[92.10009375,-87.964578125,0.676810241699219],[-7.71783197556249E-06,0.00508283936343101,0.0015183882137476,0.999985929491847],[0,0,0,0],[8.999999E+09,8.999999E+09,8.999999E+09,8.999999E+09,8.999999E+09,8.999999E+09]];
	LOCAL CONST Robtarget Tr_meulage_motif_2_P95 :=[[91.1756484375,-88.3458203125,0.684267150878906],[-7.71783197556249E-06,0.00508283936343101,0.0015183882137476,0.999985929491847],[0,0,0,0],[8.999999E+09,8.999999E+09,8.999999E+09,8.999999E+09,8.999999E+09,8.999999E+09]];
	LOCAL CONST Robtarget Tr_meulage_motif_2_P96 :=[[90.251203125,-88.7270625,0.691723999023438],[-7.71783197556249E-06,0.00508283936343101,0.0015183882137476,0.999985929491847],[0,0,0,0],[8.999999E+09,8.999999E+09,8.999999E+09,8.999999E+09,8.999999E+09,8.999999E+09]];
	LOCAL CONST Robtarget Tr_meulage_motif_2_P97 :=[[89.3267578125,-89.108296875,0.699180908203125],[-7.71783197556249E-06,0.00508283936343101,0.0015183882137476,0.999985929491847],[0,0,0,0],[8.999999E+09,8.999999E+09,8.999999E+09,8.999999E+09,8.999999E+09,8.999999E+09]];
	LOCAL CONST Robtarget Tr_meulage_motif_2_P98 :=[[88.4023125,-89.4895390625,0.706637756347656],[-7.71783197556249E-06,0.00508283936343101,0.0015183882137476,0.999985929491847],[0,0,0,0],[8.999999E+09,8.999999E+09,8.999999E+09,8.999999E+09,8.999999E+09,8.999999E+09]];
	LOCAL CONST Robtarget Tr_meulage_motif_2_P99 :=[[87.4778671875,-89.87078125,0.714094665527344],[-7.71783197556249E-06,0.00508283936343101,0.0015183882137476,0.999985929491847],[0,0,0,0],[8.999999E+09,8.999999E+09,8.999999E+09,8.999999E+09,8.999999E+09,8.999999E+09]];
	LOCAL CONST Robtarget Tr_meulage_motif_2_P100 :=[[86.553421875,-90.252015625,0.721551513671875],[-7.71783197556249E-06,0.00508283936343101,0.0015183882137476,0.999985929491847],[0,0,0,0],[8.999999E+09,8.999999E+09,8.999999E+09,8.999999E+09,8.999999E+09,8.999999E+09]];
	LOCAL CONST Robtarget Tr_meulage_motif_2_P101 :=[[85.62896875,-90.6332578125,0.729008422851563],[-7.71783197556249E-06,0.00508283936343101,0.0015183882137476,0.999985929491847],[0,0,0,0],[8.999999E+09,8.999999E+09,8.999999E+09,8.999999E+09,8.999999E+09,8.999999E+09]];
	LOCAL CONST Robtarget Tr_meulage_motif_2_P102 :=[[84.7045234375,-91.0145,0.736465270996094],[-7.71783197556249E-06,0.00508283936343101,0.0015183882137476,0.999985929491847],[0,0,0,0],[8.999999E+09,8.999999E+09,8.999999E+09,8.999999E+09,8.999999E+09,8.999999E+09]];
	LOCAL CONST Robtarget Tr_meulage_motif_2_P103 :=[[83.780078125,-91.395734375,0.743922180175781],[-7.71783197556249E-06,0.00508283936343101,0.0015183882137476,0.999985929491847],[0,0,0,0],[8.999999E+09,8.999999E+09,8.999999E+09,8.999999E+09,8.999999E+09,8.999999E+09]];
	LOCAL CONST Robtarget Tr_meulage_motif_2_P104 :=[[82.8556328125,-91.7769765625,0.751379028320313],[-7.71783197556249E-06,0.00508283936343101,0.0015183882137476,0.999985929491847],[0,0,0,0],[8.999999E+09,8.999999E+09,8.999999E+09,8.999999E+09,8.999999E+09,8.999999E+09]];
	LOCAL CONST Robtarget Tr_meulage_motif_2_P105 :=[[81.9311875,-92.15821875,0.7588359375],[-7.71783197556249E-06,0.00508283936343101,0.0015183882137476,0.999985929491847],[0,0,0,0],[8.999999E+09,8.999999E+09,8.999999E+09,8.999999E+09,8.999999E+09,8.999999E+09]];
	LOCAL CONST Robtarget Tr_meulage_motif_2_P106 :=[[81.0067421875,-92.539453125,0.766292785644531],[-7.71783197556249E-06,0.00508283936343101,0.0015183882137476,0.999985929491847],[0,0,0,0],[8.999999E+09,8.999999E+09,8.999999E+09,8.999999E+09,8.999999E+09,8.999999E+09]];
	LOCAL CONST Robtarget Tr_meulage_motif_2_P107 :=[[80.082296875,-92.9206953125,0.773749633789062],[-7.71783197556249E-06,0.00508283936343101,0.0015183882137476,0.999985929491847],[0,0,0,0],[8.999999E+09,8.999999E+09,8.999999E+09,8.999999E+09,8.999999E+09,8.999999E+09]];
	LOCAL CONST Robtarget Tr_meulage_motif_2_P108 :=[[79.1578515625,-93.3019375,0.78120654296875],[-7.71783197556249E-06,0.00508283936343101,0.0015183882137476,0.999985929491847],[0,0,0,0],[8.999999E+09,8.999999E+09,8.999999E+09,8.999999E+09,8.999999E+09,8.999999E+09]];
	LOCAL CONST Robtarget Tr_meulage_motif_2_P109 :=[[78.23340625,-93.6831796875,0.788663391113281],[-7.71783197556249E-06,0.00508283936343101,0.0015183882137476,0.999985929491847],[0,0,0,0],[8.999999E+09,8.999999E+09,8.999999E+09,8.999999E+09,8.999999E+09,8.999999E+09]];
	LOCAL CONST Robtarget Tr_meulage_motif_2_P110 :=[[77.308953125,-94.0644140625,0.796120300292969],[-7.71783197556249E-06,0.00508283936343101,0.0015183882137476,0.999985929491847],[0,0,0,0],[8.999999E+09,8.999999E+09,8.999999E+09,8.999999E+09,8.999999E+09,8.999999E+09]];
	LOCAL CONST Robtarget Tr_meulage_motif_2_P111 :=[[76.3845078125,-94.44565625,0.8035771484375],[-7.71783197556249E-06,0.00508283936343101,0.0015183882137476,0.999985929491847],[0,0,0,0],[8.999999E+09,8.999999E+09,8.999999E+09,8.999999E+09,8.999999E+09,8.999999E+09]];
	LOCAL CONST Robtarget Tr_meulage_motif_2_P112 :=[[75.4600625,-94.8268984375,0.811034057617187],[-7.71783197556249E-06,0.00508283936343101,0.0015183882137476,0.999985929491847],[0,0,0,0],[8.999999E+09,8.999999E+09,8.999999E+09,8.999999E+09,8.999999E+09,8.999999E+09]];
	LOCAL CONST Robtarget Tr_meulage_motif_2_P113 :=[[74.5356171875,-95.2081328125,0.818490905761719],[-7.71783197556249E-06,0.00508283936343101,0.0015183882137476,0.999985929491847],[0,0,0,0],[8.999999E+09,8.999999E+09,8.999999E+09,8.999999E+09,8.999999E+09,8.999999E+09]];
	LOCAL CONST Robtarget Tr_meulage_motif_2_P114 :=[[73.611171875,-95.589375,0.825947814941406],[-7.71783197556249E-06,0.00508283936343101,0.0015183882137476,0.999985929491847],[0,0,0,0],[8.999999E+09,8.999999E+09,8.999999E+09,8.999999E+09,8.999999E+09,8.999999E+09]];
	LOCAL CONST Robtarget Tr_meulage_motif_2_P115 :=[[72.6867265625,-95.9706171875,0.833404663085938],[-7.71783197556249E-06,0.00508283936343101,0.0015183882137476,0.999985929491847],[0,0,0,0],[8.999999E+09,8.999999E+09,8.999999E+09,8.999999E+09,8.999999E+09,8.999999E+09]];
	LOCAL CONST Robtarget Tr_meulage_motif_2_degg1 :=[[72.5850714399673,-96.0009853090551,-9.16603252173882],[-7.71783197556249E-06,0.00508283936343101,0.0015183882137476,0.999985929491847],[0,0,0,0],[8.999999E+09,8.999999E+09,8.999999E+09,8.999999E+09,8.999999E+09,8.999999E+09]];
	LOCAL CONST Robtarget Tr_meulage_motif_2_degg2 :=[[70.6536241118467,-96.5779796186016,-199.155339033409],[-7.71783197556249E-06,0.00508283936343101,0.0015183882137476,0.999985929491847],[0,0,0,0],[8.999999E+09,8.999999E+09,8.999999E+09,8.999999E+09,8.999999E+09,8.999999E+09]];
	LOCAL CONST Robtarget Tr_meulage_bavure_App1 :=[[338.704090609516,98.7594988633749,39.5940069054088],[0.237070036667954,-0.257628036320879,-0.68928427529211,0.634281310185578],[0,0,0,0],[8.999999E+09,8.999999E+09,8.999999E+09,8.999999E+09,8.999999E+09,8.999999E+09]];
	LOCAL CONST Robtarget Tr_meulage_bavure_App2 :=[[214.513517811726,-44.1677143146438,23.8297003452704],[0.237070036667954,-0.257628036320879,-0.68928427529211,0.634281310185578],[0,0,0,0],[8.999999E+09,8.999999E+09,8.999999E+09,8.999999E+09,8.999999E+09,8.999999E+09]];
	LOCAL CONST Robtarget Tr_meulage_bavure_P0 :=[[207.977171875,-51.69019921875,23],[0.237070036667954,-0.257628036320879,-0.68928427529211,0.634281310185578],[0,0,0,0],[8.999999E+09,8.999999E+09,8.999999E+09,8.999999E+09,8.999999E+09,8.999999E+09]];
	LOCAL CONST Robtarget Tr_meulage_bavure_P1 :=[[206.08234375,-48.4886328125,23],[0.231785854990408,-0.251833962519259,-0.691348546178018,0.636311370671431],[0,0,0,0],[8.999999E+09,8.999999E+09,8.999999E+09,8.999999E+09,8.999999E+09,8.999999E+09]];
	LOCAL CONST Robtarget Tr_meulage_bavure_P2 :=[[204.130609375,-46.47016796875,23],[0.216488884662801,-0.235071780299825,-0.697010963315473,0.641910848905176],[0,0,0,0],[8.999999E+09,8.999999E+09,8.999999E+09,8.999999E+09,8.999999E+09,8.999999E+09]];
	LOCAL CONST Robtarget Tr_meulage_bavure_P3 :=[[203.69896875,-45.613921875,23],[0.192788956393482,-0.209131813375552,-0.704882013414004,0.649798161041092],[0,0,0,0],[8.999999E+09,8.999999E+09,8.999999E+09,8.999999E+09,8.999999E+09,8.999999E+09]];
	LOCAL CONST Robtarget Tr_meulage_bavure_P4 :=[[203.31628125,-44.69117578125,23],[0.163255625326789,-0.176859349674191,-0.713200051417095,0.658341900451911],[0,0,0,0],[8.999999E+09,8.999999E+09,8.999999E+09,8.999999E+09,8.999999E+09,8.999999E+09]];
	LOCAL CONST Robtarget Tr_meulage_bavure_P5 :=[[202.150703125,-43.93252734375,23],[0.131034075209159,-0.141719879494531,-0.720439369423193,0.666117603637112],[0,0,0,0],[8.999999E+09,8.999999E+09,8.999999E+09,8.999999E+09,8.999999E+09,8.999999E+09]];
	LOCAL CONST Robtarget Tr_meulage_bavure_P6 :=[[200.419859375,-42.90380859375,23],[0.0992738652180014,-0.107166948106979,-0.725736560080676,0.672284456372733],[0,0,0,0],[8.999999E+09,8.999999E+09,8.999999E+09,8.999999E+09,8.999999E+09,8.999999E+09]];
	LOCAL CONST Robtarget Tr_meulage_bavure_P7 :=[[198.04265625,-42.7425859375,23],[0.070572316930657,-0.0760244077419609,-0.728944442786691,0.676668188140187],[0,0,0,0],[8.999999E+09,8.999999E+09,8.999999E+09,8.999999E+09,8.999999E+09,8.999999E+09]];
	LOCAL CONST Robtarget Tr_meulage_bavure_P8 :=[[197.17828125,-42.69424609375,23],[0.0466490069803766,-0.0501411146580529,-0.730423260552647,0.679552499231835],[0,0,0,0],[8.999999E+09,8.999999E+09,8.999999E+09,8.999999E+09,8.999999E+09,8.999999E+09]];
	LOCAL CONST Robtarget Tr_meulage_bavure_P9 :=[[196.593203125,-42.76303125,23],[0.0282922727868155,-0.0303405010582799,-0.730732536258324,0.681402202630404],[0,0,0,0],[8.999999E+09,8.999999E+09,8.999999E+09,8.999999E+09,8.999999E+09,8.999999E+09]];
	LOCAL CONST Robtarget Tr_meulage_bavure_P10 :=[[195.3330625,-42.9101875,23],[0.0155330463889182,-0.0166191395142733,-0.730386926946294,0.682654719179201],[0,0,0,0],[8.999999E+09,8.999999E+09,8.999999E+09,8.999999E+09,8.999999E+09,8.999999E+09]];
	LOCAL CONST Robtarget Tr_meulage_bavure_P11 :=[[194.0414375,-42.98870703125,23],[0.00787853097781009,-0.00841034895474212,-0.729755879459697,0.683610672220742],[0,0,0,0],[8.999999E+09,8.999999E+09,8.999999E+09,8.999999E+09,8.999999E+09,8.999999E+09]];
	LOCAL CONST Robtarget Tr_meulage_bavure_P12 :=[[191.22246875,-43.17755078125,23],[0.00454087568737026,-0.00483683003246043,-0.729043591690291,0.684435115214401],[0,0,0,0],[8.999999E+09,8.999999E+09,8.999999E+09,8.999999E+09,8.999999E+09,8.999999E+09]];
	LOCAL CONST Robtarget Tr_meulage_bavure_P13 :=[[187.99846875,-43.3063984375,23],[0.00460825153360559,-0.00489854980895224,-0.728342920317329,0.685179800235819],[0,0,0,0],[8.999999E+09,8.999999E+09,8.999999E+09,8.999999E+09,8.999999E+09,8.999999E+09]];
	LOCAL CONST Robtarget Tr_meulage_bavure_P14 :=[[185.297671875,-43.3160078125,23],[0.00721178706639714,-0.00765162620458669,-0.727672749199787,0.685843869124569],[0,0,0,0],[8.999999E+09,8.999999E+09,8.999999E+09,8.999999E+09,8.999999E+09,8.999999E+09]];
	LOCAL CONST Robtarget Tr_meulage_bavure_P15 :=[[183.1435625,-43.26251171875,23],[0.0116459139289,-0.0123350411953757,-0.727021716176972,0.686404868612221],[0,0,0,0],[8.999999E+09,8.999999E+09,8.999999E+09,8.999999E+09,8.999999E+09,8.999999E+09]];
	LOCAL CONST Robtarget Tr_meulage_bavure_P16 :=[[181.0938125,-43.12933203125,23],[0.0174146518227317,-0.0184172452497901,-0.726374138490383,0.686831963373615],[0,0,0,0],[8.999999E+09,8.999999E+09,8.999999E+09,8.999999E+09,8.999999E+09,8.999999E+09]];
	LOCAL CONST Robtarget Tr_meulage_bavure_P17 :=[[179.112125,-42.960359375,23],[0.024261191892774,-0.0256242088293737,-0.725703782479072,0.687101749805208],[0,0,0,0],[8.999999E+09,8.999999E+09,8.999999E+09,8.999999E+09,8.999999E+09,8.999999E+09]];
	LOCAL CONST Robtarget Tr_meulage_bavure_P18 :=[[176.1563125,-42.7535078125,23],[0.0320223457964327,-0.0337834988106105,-0.724984404104576,0.68719055463746],[0,0,0,0],[8.999999E+09,8.999999E+09,8.999999E+09,8.999999E+09,8.999999E+09,8.999999E+09]];
	LOCAL CONST Robtarget Tr_meulage_bavure_P19 :=[[173.821171875,-42.483703125,23],[0.0405378300180767,-0.0427274170241108,-0.724191083502512,0.687079563622242],[0,0,0,0],[8.999999E+09,8.999999E+09,8.999999E+09,8.999999E+09,8.999999E+09,8.999999E+09]];
	LOCAL CONST Robtarget Tr_meulage_bavure_P20 :=[[170.8773125,-42.02716015625,23],[0.0495921326273582,-0.0522305765020709,-0.723302644831425,0.686764785963577],[0,0,0,0],[8.999999E+09,8.999999E+09,8.999999E+09,8.999999E+09,8.999999E+09,8.999999E+09]];
	LOCAL CONST Robtarget Tr_meulage_bavure_P21 :=[[168.39421875,-41.59423828125,23],[0.0589299198174011,-0.0620268729941979,-0.722315506136558,0.686250858776558],[0,0,0,0],[8.999999E+09,8.999999E+09,8.999999E+09,8.999999E+09,8.999999E+09,8.999999E+09]];
	LOCAL CONST Robtarget Tr_meulage_bavure_P22 :=[[166.971625,-41.32940625,23],[0.0683338371567196,-0.0718894708503375,-0.72122988592947,0.685558051752338],[0,0,0,0],[8.999999E+09,8.999999E+09,8.999999E+09,8.999999E+09,8.999999E+09,8.999999E+09]];
	LOCAL CONST Robtarget Tr_meulage_bavure_P23 :=[[164.19171875,-40.64562890625,23],[0.0776601128749892,-0.0816686256947137,-0.720050746025756,0.684708745082997],[0,0,0,0],[8.999999E+09,8.999999E+09,8.999999E+09,8.999999E+09,8.999999E+09,8.999999E+09]];
	LOCAL CONST Robtarget Tr_meulage_bavure_P24 :=[[161.096921875,-39.8893125,23],[0.0868334142276125,-0.0912864262493833,-0.71878457332933,0.683721788229661],[0,0,0,0],[8.999999E+09,8.999999E+09,8.999999E+09,8.999999E+09,8.999999E+09,8.999999E+09]];
	LOCAL CONST Robtarget Tr_meulage_bavure_P25 :=[[158.411921875,-39.136140625,23],[0.0958208372696551,-0.100707260403892,-0.717430431693702,0.682619945889858],[0,0,0,0],[8.999999E+09,8.999999E+09,8.999999E+09,8.999999E+09,8.999999E+09,8.999999E+09]];
	LOCAL CONST Robtarget Tr_meulage_bavure_P26 :=[[156.437921875,-38.54827734375,23],[0.104588753529082,-0.109894933624012,-0.715993917086247,0.681422781314581],[0,0,0,0],[8.999999E+09,8.999999E+09,8.999999E+09,8.999999E+09,8.999999E+09,8.999999E+09]];
	LOCAL CONST Robtarget Tr_meulage_bavure_P27 :=[[152.714359375,-37.2186875,23],[0.113093838547092,-0.118802269370906,-0.714484038979192,0.680153190479165],[0,0,0,0],[8.999999E+09,8.999999E+09,8.999999E+09,8.999999E+09,8.999999E+09,8.999999E+09]];
	LOCAL CONST Robtarget Tr_meulage_bavure_P28 :=[[151.92065625,-36.92523046875,23],[0.121294937123283,-0.127384080145817,-0.712912742386012,0.678834483579995],[0,0,0,0],[8.999999E+09,8.999999E+09,8.999999E+09,8.999999E+09,8.999999E+09,8.999999E+09]];
	LOCAL CONST Robtarget Tr_meulage_bavure_P29 :=[[151.537046875,-36.71096875,23],[0.129192351412326,-0.135638300828311,-0.711285970603551,0.677483472645294],[0,0,0,0],[8.999999E+09,8.999999E+09,8.999999E+09,8.999999E+09,8.999999E+09,8.999999E+09]];
	LOCAL CONST Robtarget Tr_meulage_bavure_P30 :=[[148.450859375,-35.4978046875,23],[0.13683324908827,-0.14361110153132,-0.709598481258918,0.676108355854256],[0,0,0,0],[8.999999E+09,8.999999E+09,8.999999E+09,8.999999E+09,8.999999E+09,8.999999E+09]];
	LOCAL CONST Robtarget Tr_meulage_bavure_P31 :=[[145.888421875,-34.38015625,23],[0.144269217550455,-0.15135526385495,-0.707847140925119,0.674707641912342],[0,0,0,0],[8.999999E+09,8.999999E+09,8.999999E+09,8.999999E+09,8.999999E+09,8.999999E+09]];
	LOCAL CONST Robtarget Tr_meulage_bavure_P32 :=[[144.439265625,-33.7287890625,23],[0.151565124419104,-0.158937623297997,-0.706023513178855,0.673273825273783],[0,0,0,0],[8.999999E+09,8.999999E+09,8.999999E+09,8.999999E+09,8.999999E+09,8.999999E+09]];
	LOCAL CONST Robtarget Tr_meulage_bavure_P33 :=[[142.42290625,-32.713654296875,23],[0.158768704734715,-0.166404184105213,-0.704115046835644,0.671806628970553],[0,0,0,0],[8.999999E+09,8.999999E+09,8.999999E+09,8.999999E+09,8.999999E+09,8.999999E+09]];
	LOCAL CONST Robtarget Tr_meulage_bavure_P34 :=[[139.73553125,-31.357818359375,23],[0.165910260432823,-0.173784825882325,-0.702116557079152,0.670302140867446],[0,0,0,0],[8.999999E+09,8.999999E+09,8.999999E+09,8.999999E+09,8.999999E+09,8.999999E+09]];
	LOCAL CONST Robtarget Tr_meulage_bavure_P35 :=[[138.7085625,-30.780517578125,23],[0.173041287004779,-0.181134780003364,-0.700021338015115,0.668742873448675],[0,0,0,0],[8.999999E+09,8.999999E+09,8.999999E+09,8.999999E+09,8.999999E+09,8.999999E+09]];
	LOCAL CONST Robtarget Tr_meulage_bavure_P36 :=[[134.67565625,-28.541931640625,23],[0.180236872994927,-0.188532379524369,-0.69781034589641,0.667106387800194],[0,0,0,0],[8.999999E+09,8.999999E+09,8.999999E+09,8.999999E+09,8.999999E+09,8.999999E+09]];
	LOCAL CONST Robtarget Tr_meulage_bavure_P37 :=[[133.343328125,-27.7184140625,23],[0.187615182704433,-0.196101037819058,-0.695448414094891,0.665354363867835],[0,0,0,0],[8.999999E+09,8.999999E+09,8.999999E+09,8.999999E+09,8.999999E+09,8.999999E+09]];
	LOCAL CONST Robtarget Tr_meulage_bavure_P38 :=[[129.1232265625,-25.053009765625,23],[0.195288037768213,-0.203956967478761,-0.692895829816471,0.663445179908975],[0,0,0,0],[8.999999E+09,8.999999E+09,8.999999E+09,8.999999E+09,8.999999E+09,8.999999E+09]];
	LOCAL CONST Robtarget Tr_meulage_bavure_P39 :=[[128.160890625,-24.394134765625,23],[0.203343988155317,-0.212195802010507,-0.690119731796249,0.661331172617533],[0,0,0,0],[8.999999E+09,8.999999E+09,8.999999E+09,8.999999E+09,8.999999E+09,8.999999E+09]];
	LOCAL CONST Robtarget Tr_meulage_bavure_P40 :=[[127.2111171875,-23.759185546875,23],[0.211848646914484,-0.220887225221036,-0.687085715997349,0.658970563384332],[0,0,0,0],[8.999999E+09,8.999999E+09,8.999999E+09,8.999999E+09,8.999999E+09,8.999999E+09]];
	LOCAL CONST Robtarget Tr_meulage_bavure_P41 :=[[123.2999296875,-20.87222265625,23],[0.220808575365934,-0.230038130032332,-0.683772978209739,0.6563387433683],[0,0,0,0],[8.999999E+09,8.999999E+09,8.999999E+09,8.999999E+09,8.999999E+09,8.999999E+09]];
	LOCAL CONST Robtarget Tr_meulage_bavure_P42 :=[[121.436828125,-19.447662109375,23],[0.230198366107411,-0.23962724235316,-0.68017614654288,0.653412508785818],[0,0,0,0],[8.999999E+09,8.999999E+09,8.999999E+09,8.999999E+09,8.999999E+09,8.999999E+09]];
	LOCAL CONST Robtarget Tr_meulage_bavure_P43 :=[[118.5504765625,-16.96597265625,23],[0.239959075245837,-0.249594773558409,-0.676296856801556,0.650188167148423],[0,0,0,0],[8.999999E+09,8.999999E+09,8.999999E+09,8.999999E+09,8.999999E+09,8.999999E+09]];
	LOCAL CONST Robtarget Tr_meulage_bavure_P44 :=[[116.69665625,-15.358458984375,23],[0.249992260334041,-0.25983909548538,-0.672153515994317,0.646681656742244],[0,0,0,0],[8.999999E+09,8.999999E+09,8.999999E+09,8.999999E+09,8.999999E+09,8.999999E+09]];
	LOCAL CONST Robtarget Tr_meulage_bavure_P45 :=[[115.805484375,-14.479796875,23],[0.260146575466534,-0.270204155814859,-0.667792567830207,0.642935890897493],[0,0,0,0],[8.999999E+09,8.999999E+09,8.999999E+09,8.999999E+09,8.999999E+09,8.999999E+09]];
	LOCAL CONST Robtarget Tr_meulage_bavure_P46 :=[[115.2398046875,-13.865478515625,23],[0.270223142651443,-0.280485320363437,-0.663291804663466,0.639023802453774],[0,0,0,0],[8.999999E+09,8.999999E+09,8.999999E+09,8.999999E+09,8.999999E+09,8.999999E+09]];
	LOCAL CONST Robtarget Tr_meulage_bavure_P47 :=[[114.0506015625,-12.599853515625,23],[0.280010651495607,-0.290461981648059,-0.658745904080689,0.635043074226469],[0,0,0,0],[8.999999E+09,8.999999E+09,8.999999E+09,8.999999E+09,8.999999E+09,8.999999E+09]];
	LOCAL CONST Robtarget Tr_meulage_bavure_P48 :=[[111.224703125,-9.3840634765625,23],[0.289301971033488,-0.299917545270759,-0.654262907191103,0.631105287466955],[0,0,0,0],[8.999999E+09,8.999999E+09,8.999999E+09,8.999999E+09,8.999999E+09,8.999999E+09]];
	LOCAL CONST Robtarget Tr_meulage_bavure_P49 :=[[109.7358671875,-7.595947265625,23],[0.29792002749699,-0.308663390899651,-0.649948173460453,0.62732602381054],[0,0,0,0],[8.999999E+09,8.999999E+09,8.999999E+09,8.999999E+09,8.999999E+09,8.999999E+09]];
	LOCAL CONST Robtarget Tr_meulage_bavure_P50 :=[[107.117859375,-4.238861328125,23],[0.305733221456827,-0.316559287196041,-0.645896294280843,0.623807175352961],[0,0,0,0],[8.999999E+09,8.999999E+09,8.999999E+09,8.999999E+09,8.999999E+09,8.999999E+09]];
	LOCAL CONST Robtarget Tr_meulage_bavure_P51 :=[[105.9093359375,-2.58413696289063,23],[0.312660814049253,-0.323511640362385,-0.642177296892776,0.620638182247584],[0,0,0,0],[8.999999E+09,8.999999E+09,8.999999E+09,8.999999E+09,8.999999E+09,8.999999E+09]];
	LOCAL CONST Robtarget Tr_meulage_bavure_P52 :=[[104.580625,-0.66387939453125,23],[0.318673279166636,-0.329483359408488,-0.638838218145137,0.61787845734839],[0,0,0,0],[8.999999E+09,8.999999E+09,8.999999E+09,8.999999E+09,8.999999E+09,8.999999E+09]];
	LOCAL CONST Robtarget Tr_meulage_bavure_P53 :=[[104.26040625,-0.150238037109375,23],[0.323842647390335,-0.33453857832565,-0.635865909530693,0.615535883957854],[0,0,0,0],[8.999999E+09,8.999999E+09,8.999999E+09,8.999999E+09,8.999999E+09,8.999999E+09]];
	LOCAL CONST Robtarget Tr_meulage_bavure_P54 :=[[101.7081328125,3.79440307617188,23],[0.3283697541188,-0.338875835757285,-0.633170367797755,0.613540347379548],[0,0,0,0],[8.999999E+09,8.999999E+09,8.999999E+09,8.999999E+09,8.999999E+09,8.999999E+09]];
	LOCAL CONST Robtarget Tr_meulage_bavure_P55 :=[[99.1396796875,7.8708798828125,23],[0.332587507577216,-0.342829250764221,-0.63057767924243,0.611739687338699],[0,0,0,0],[8.999999E+09,8.999999E+09,8.999999E+09,8.999999E+09,8.999999E+09,8.999999E+09]];
	LOCAL CONST Robtarget Tr_meulage_bavure_P56 :=[[97.95065625,9.6949765625,23],[0.336882002635063,-0.346786489991634,-0.627872086071277,0.609939579132536],[0,0,0,0],[8.999999E+09,8.999999E+09,8.999999E+09,8.999999E+09,8.999999E+09,8.999999E+09]];
	LOCAL CONST Robtarget Tr_meulage_bavure_P57 :=[[97.205078125,11.0410458984375,23],[0.341580260223243,-0.3510749834348,-0.624861184146566,0.607961990899948],[0,0,0,0],[8.999999E+09,8.999999E+09,8.999999E+09,8.999999E+09,8.999999E+09,8.999999E+09]];
	LOCAL CONST Robtarget Tr_meulage_bavure_P58 :=[[96.785,11.8498232421875,23],[0.346850169899341,-0.355855764716803,-0.621433959047775,0.605707411957974],[0,0,0,0],[8.999999E+09,8.999999E+09,8.999999E+09,8.999999E+09,8.999999E+09,8.999999E+09]];
	LOCAL CONST Robtarget Tr_meulage_bavure_P59 :=[[95.9808359375,13.22998046875,23],[0.352631821301647,-0.361058330833286,-0.61761006618864,0.603196059738314],[0,0,0,0],[8.999999E+09,8.999999E+09,8.999999E+09,8.999999E+09,8.999999E+09,8.999999E+09]];
	LOCAL CONST Robtarget Tr_meulage_bavure_P60 :=[[94.8823515625,15.3327333984375,23],[0.358676059646391,-0.366423028917287,-0.613528287113346,0.600556982331721],[0,0,0,0],[8.999999E+09,8.999999E+09,8.999999E+09,8.999999E+09,8.999999E+09,8.999999E+09]];
	LOCAL CONST Robtarget Tr_meulage_bavure_P61 :=[[94.038546875,16.99914453125,23],[0.364632666113741,-0.371587594022814,-0.609400213481013,0.597994196109308],[0,0,0,0],[8.999999E+09,8.999999E+09,8.999999E+09,8.999999E+09,8.999999E+09,8.999999E+09]];
	LOCAL CONST Robtarget Tr_meulage_bavure_P62 :=[[90.59884375,24.24755859375,23],[0.370138252458813,-0.37618505468689,-0.605463784598971,0.595731553836162],[0,0,0,0],[8.999999E+09,8.999999E+09,8.999999E+09,8.999999E+09,8.999999E+09,8.999999E+09]];
	LOCAL CONST Robtarget Tr_meulage_bavure_P63 :=[[90.4949375,24.4801640625,23],[0.37488055040896,-0.379909891387611,-0.601939703649603,0.593971077175612],[0,0,0,0],[8.999999E+09,8.999999E+09,8.999999E+09,8.999999E+09,8.999999E+09,8.999999E+09]];
	LOCAL CONST Robtarget Tr_meulage_bavure_P64 :=[[87.2562578125,32.08935546875,23],[0.378673730413387,-0.382586922955739,-0.598972053967407,0.592845621426131],[0,0,0,0],[8.999999E+09,8.999999E+09,8.999999E+09,8.999999E+09,8.999999E+09,8.999999E+09]];
	LOCAL CONST Robtarget Tr_meulage_bavure_P65 :=[[87.0634453125,32.55319140625,23],[0.38149227020855,-0.384212667528063,-0.596601527263637,0.592377321939988],[0,0,0,0],[8.999999E+09,8.999999E+09,8.999999E+09,8.999999E+09,8.999999E+09,8.999999E+09]];
	LOCAL CONST Robtarget Tr_meulage_bavure_P66 :=[[86.7218359375,33.27237109375,23],[0.383484825486142,-0.384957969584776,-0.594747346104907,0.592471387137134],[0,0,0,0],[8.999999E+09,8.999999E+09,8.999999E+09,8.999999E+09,8.999999E+09,8.999999E+09]];
	LOCAL CONST Robtarget Tr_meulage_bavure_P67 :=[[84.9730546875,36.9846796875,23],[0.384928203554605,-0.385125953655032,-0.593240929180389,0.592936318566096],[0,0,0,0],[8.999999E+09,8.999999E+09,8.999999E+09,8.999999E+09,8.999999E+09,8.999999E+09]];
	LOCAL CONST Robtarget Tr_meulage_bavure_P68 :=[[84.3369453125,38.347078125,23],[0.386125187380856,-0.385041592383358,-0.591893434564505,0.593559157897863],[0,0,0,0],[8.999999E+09,8.999999E+09,8.999999E+09,8.999999E+09,8.999999E+09,8.999999E+09]];
	LOCAL CONST Robtarget Tr_meulage_bavure_P69 :=[[84.2352265625,38.57379296875,23],[0.387303414207436,-0.384949718441005,-0.590564063612056,0.594174945942245],[0,0,0,0],[8.999999E+09,8.999999E+09,8.999999E+09,8.999999E+09,8.999999E+09,8.999999E+09]];
	LOCAL CONST Robtarget Tr_meulage_bavure_P70 :=[[81.203640625,45.7033984375,23],[0.388529428696597,-0.384935767637602,-0.589218441508191,0.594719232929796],[0,0,0,0],[8.999999E+09,8.999999E+09,8.999999E+09,8.999999E+09,8.999999E+09,8.999999E+09]];
	LOCAL CONST Robtarget Tr_meulage_bavure_P71 :=[[78.802765625,51.43176171875,23],[0.389745197294745,-0.384963800490539,-0.587904112662146,0.595206105321925],[0,0,0,0],[8.999999E+09,8.999999E+09,8.999999E+09,8.999999E+09,8.999999E+09,8.999999E+09]];
	LOCAL CONST Robtarget Tr_meulage_bavure_P72 :=[[77.2335546875,55.184328125,23],[0.390849057815693,-0.384952373300406,-0.586695273697821,0.595682247608244],[0,0,0,0],[8.999999E+09,8.999999E+09,8.999999E+09,8.999999E+09,8.999999E+09,8.999999E+09]];
	LOCAL CONST Robtarget Tr_meulage_bavure_P73 :=[[76.2354140625,57.48068359375,23],[0.391789739118034,-0.384867875904665,-0.585632181367356,0.596164798160179],[0,0,0,0],[8.999999E+09,8.999999E+09,8.999999E+09,8.999999E+09,8.999999E+09,8.999999E+09]];
	LOCAL CONST Robtarget Tr_meulage_bavure_P74 :=[[75.3550390625,59.70236328125,23],[0.392621634591246,-0.384781423966826,-0.584687225606464,0.596600667141411],[0,0,0,0],[8.999999E+09,8.999999E+09,8.999999E+09,8.999999E+09,8.999999E+09,8.999999E+09]];
	LOCAL CONST Robtarget Tr_meulage_bavure_P75 :=[[72.003109375,67.565609375,23],[0.393479692981755,-0.384844633268658,-0.583782108431558,0.596880883703358],[0,0,0,0],[8.999999E+09,8.999999E+09,8.999999E+09,8.999999E+09,8.999999E+09,8.999999E+09]];
	LOCAL CONST Robtarget Tr_meulage_bavure_P76 :=[[71.67584375,68.4326484375,23],[0.394518281815651,-0.385221447895635,-0.582823416205807,0.596889124475066],[0,0,0,0],[8.999999E+09,8.999999E+09,8.999999E+09,8.999999E+09,8.999999E+09,8.999999E+09]];
	LOCAL CONST Robtarget Tr_meulage_bavure_P77 :=[[70.4950546875,71.100859375,23],[0.395823771792468,-0.386002344496033,-0.581757689164558,0.59655990715557],[0,0,0,0],[8.999999E+09,8.999999E+09,8.999999E+09,8.999999E+09,8.999999E+09,8.999999E+09]];
	LOCAL CONST Robtarget Tr_meulage_bavure_P78 :=[[69.626375,73.06378125,23],[0.397363389346432,-0.387162490694565,-0.580607246899425,0.595904998681978],[0,0,0,0],[8.999999E+09,8.999999E+09,8.999999E+09,8.999999E+09,8.999999E+09,8.999999E+09]];
	LOCAL CONST Robtarget Tr_meulage_bavure_P79 :=[[68.3869609375,76.0791953125,23],[0.398982289671604,-0.388556512090641,-0.579471937424726,0.595020372069389],[0,0,0,0],[8.999999E+09,8.999999E+09,8.999999E+09,8.999999E+09,8.999999E+09,8.999999E+09]];
	LOCAL CONST Robtarget Tr_meulage_bavure_P80 :=[[67.6337890625,78.0066796875,23],[0.400453292643468,-0.389964709530787,-0.578498224027534,0.594057649162573],[0,0,0,0],[8.999999E+09,8.999999E+09,8.999999E+09,8.999999E+09,8.999999E+09,8.999999E+09]];
	LOCAL CONST Robtarget Tr_meulage_bavure_P81 :=[[66.77353125,80.39465625,23],[0.401561564819311,-0.39117388370929,-0.577824931299211,0.593169158952755],[0,0,0,0],[8.999999E+09,8.999999E+09,8.999999E+09,8.999999E+09,8.999999E+09,8.999999E+09]];
	LOCAL CONST Robtarget Tr_meulage_bavure_P82 :=[[63.83282421875,87.6394375,23],[0.40219044665569,-0.39206368878238,-0.577527587277447,0.592444760708322],[0,0,0,0],[8.999999E+09,8.999999E+09,8.999999E+09,8.999999E+09,8.999999E+09,8.999999E+09]];
	LOCAL CONST Robtarget Tr_meulage_bavure_P83 :=[[63.5959453125,88.1963203125,23],[0.402365813126573,-0.392644529911255,-0.577584825859143,0.591884950387341],[0,0,0,0],[8.999999E+09,8.999999E+09,8.999999E+09,8.999999E+09,8.999999E+09,8.999999E+09]];
	LOCAL CONST Robtarget Tr_meulage_bavure_P84 :=[[61.52261328125,93.64325,23],[0.402246963462192,-0.393054834981874,-0.577885284825699,0.591399927853174],[0,0,0,0],[8.999999E+09,8.999999E+09,8.999999E+09,8.999999E+09,8.999999E+09,8.999999E+09]];
	LOCAL CONST Robtarget Tr_meulage_bavure_P85 :=[[61.46926953125,93.8003515625,23],[0.402061858140275,-0.393501175358449,-0.578271162313339,0.590851546547091],[0,0,0,0],[8.999999E+09,8.999999E+09,8.999999E+09,8.999999E+09,8.999999E+09,8.999999E+09]];
	LOCAL CONST Robtarget Tr_meulage_bavure_P86 :=[[61.32934375,94.19915625,23],[0.402017278771884,-0.394163592011568,-0.578594696817019,0.59012316266743],[0,0,0,0],[8.999999E+09,8.999999E+09,8.999999E+09,8.999999E+09,8.999999E+09,8.999999E+09]];
	LOCAL CONST Robtarget Tr_meulage_bavure_P87 :=[[60.29598828125,96.8335234375,23],[0.402218754497096,-0.395123107741951,-0.578773968926787,0.589167629925373],[0,0,0,0],[8.999999E+09,8.999999E+09,8.999999E+09,8.999999E+09,8.999999E+09,8.999999E+09]];
	LOCAL CONST Robtarget Tr_meulage_bavure_P88 :=[[60.0941171875,97.3070703125,23],[0.402641779477194,-0.396332882168882,-0.578813006748802,0.588026655135255],[0,0,0,0],[8.999999E+09,8.999999E+09,8.999999E+09,8.999999E+09,8.999999E+09,8.999999E+09]];
	LOCAL CONST Robtarget Tr_meulage_bavure_P89 :=[[58.83993359375,100.0791328125,23],[0.403154652909552,-0.39764031856444,-0.578788759756832,0.586815196180618],[0,0,0,0],[8.999999E+09,8.999999E+09,8.999999E+09,8.999999E+09,8.999999E+09,8.999999E+09]];
	LOCAL CONST Robtarget Tr_meulage_bavure_P90 :=[[55.4352734375,108.492125,23],[0.403578062024321,-0.39884605509307,-0.578813346375003,0.585680529168897],[0,0,0,0],[8.999999E+09,8.999999E+09,8.999999E+09,8.999999E+09,8.999999E+09,8.999999E+09]];
	LOCAL CONST Robtarget Tr_meulage_bavure_P91 :=[[55.205015625,109.082546875,23],[0.403747926175968,-0.39976447559639,-0.578991311496299,0.584760666744561],[0,0,0,0],[8.999999E+09,8.999999E+09,8.999999E+09,8.999999E+09,8.999999E+09,8.999999E+09]];
	LOCAL CONST Robtarget Tr_meulage_bavure_P92 :=[[53.28241015625,113.8409140625,23],[0.403544594542811,-0.400255545512128,-0.57939942408323,0.584160565148049],[0,0,0,0],[8.999999E+09,8.999999E+09,8.999999E+09,8.999999E+09,8.999999E+09,8.999999E+09]];
	LOCAL CONST Robtarget Tr_meulage_bavure_P93 :=[[53.1260390625,114.2705390625,23],[0.402909213384753,-0.400239779131402,-0.580072793727574,0.583941640018601],[0,0,0,0],[8.999999E+09,8.999999E+09,8.999999E+09,8.999999E+09,8.999999E+09,8.999999E+09]];
	LOCAL CONST Robtarget Tr_meulage_bavure_P94 :=[[52.9638671875,114.6949453125,23],[0.401840370440164,-0.399694830501164,-0.581005398844197,0.58412420397468],[0,0,0,0],[8.999999E+09,8.999999E+09,8.999999E+09,8.999999E+09,8.999999E+09,8.999999E+09]];
	LOCAL CONST Robtarget Tr_meulage_bavure_P95 :=[[52.85201953125,115.028046875,23],[0.40038981768968,-0.398662794800758,-0.58215689293861,0.584678819469405],[0,0,0,0],[8.999999E+09,8.999999E+09,8.999999E+09,8.999999E+09,8.999999E+09,8.999999E+09]];
	LOCAL CONST Robtarget Tr_meulage_bavure_P96 :=[[50.93145703125,120.3733515625,23],[0.398674155091923,-0.397248663458074,-0.583440239298452,0.585533862906221],[0,0,0,0],[8.999999E+09,8.999999E+09,8.999999E+09,8.999999E+09,8.999999E+09,8.999999E+09]];
	LOCAL CONST Robtarget Tr_meulage_bavure_P97 :=[[49.4595625,123.8785078125,23],[0.396865612185791,-0.395612814457569,-0.58473040337493,0.586582084852879],[0,0,0,0],[8.999999E+09,8.999999E+09,8.999999E+09,8.999999E+09,8.999999E+09,8.999999E+09]];
	LOCAL CONST Robtarget Tr_meulage_bavure_P98 :=[[48.0731796875,127.1129765625,23],[0.39516611765387,-0.393955143802488,-0.585888012363721,0.587688966289497],[0,0,0,0],[8.999999E+09,8.999999E+09,8.999999E+09,8.999999E+09,8.999999E+09,8.999999E+09]];
	LOCAL CONST Robtarget Tr_meulage_bavure_P99 :=[[46.68155078125,130.5522734375,23],[0.393771727239107,-0.392468832877065,-0.58678028300831,0.588728240803797],[0,0,0,0],[8.999999E+09,8.999999E+09,8.999999E+09,8.999999E+09,8.999999E+09,8.999999E+09]];
	LOCAL CONST Robtarget Tr_meulage_bavure_P100 :=[[44.55901953125,136.1095,23],[0.392836515491265,-0.391310509333222,-0.587307433274468,0.589597774930173],[0,0,0,0],[8.999999E+09,8.999999E+09,8.999999E+09,8.999999E+09,8.999999E+09,8.999999E+09]];
	LOCAL CONST Robtarget Tr_meulage_bavure_P101 :=[[43.58938671875,138.355953125,23],[0.392455130462378,-0.390570534114205,-0.587407744947728,0.590242127970317],[0,0,0,0],[8.999999E+09,8.999999E+09,8.999999E+09,8.999999E+09,8.999999E+09,8.999999E+09]];
	LOCAL CONST Robtarget Tr_meulage_bavure_P102 :=[[43.38986328125,138.828671875,23],[0.392640879212185,-0.390263276029817,-0.587075549999176,0.590652193720739],[0,0,0,0],[8.999999E+09,8.999999E+09,8.999999E+09,8.999999E+09,8.999999E+09,8.999999E+09]];
	LOCAL CONST Robtarget Tr_meulage_bavure_P103 :=[[43.13546875,139.410640625,23],[0.39333134439505,-0.39033421031551,-0.5863571894379,0.590859462282053],[0,0,0,0],[8.999999E+09,8.999999E+09,8.999999E+09,8.999999E+09,8.999999E+09,8.999999E+09]];
	LOCAL CONST Robtarget Tr_meulage_bavure_P104 :=[[41.83837890625,142.429078125,23],[0.394401470276973,-0.390659532340961,-0.585336491736897,0.590943145721859],[0,0,0,0],[8.999999E+09,8.999999E+09,8.999999E+09,8.999999E+09,8.999999E+09,8.999999E+09]];
	LOCAL CONST Robtarget Tr_meulage_bavure_P105 :=[[40.58508203125,145.431,23],[0.39568257567676,-0.391077217607291,-0.584127755420104,0.591006492791929],[0,0,0,0],[8.999999E+09,8.999999E+09,8.999999E+09,8.999999E+09,8.999999E+09,8.999999E+09]];
	LOCAL CONST Robtarget Tr_meulage_bavure_P106 :=[[38.96469140625,149.5609375,23],[0.396997197600797,-0.391422719448751,-0.582853467909821,0.591154222468175],[0,0,0,0],[8.999999E+09,8.999999E+09,8.999999E+09,8.999999E+09,8.999999E+09,8.999999E+09]];
	LOCAL CONST Robtarget Tr_meulage_bavure_P107 :=[[37.887359375,152.354859375,23],[0.398189726348813,-0.391555245578241,-0.581622122704243,0.591477081442241],[0,0,0,0],[8.999999E+09,8.999999E+09,8.999999E+09,8.999999E+09,8.999999E+09,8.999999E+09]];
	LOCAL CONST Robtarget Tr_meulage_bavure_P108 :=[[36.45703125,155.921328125,23],[0.399156115313363,-0.391394084579676,-0.580511067770343,0.592023619765393],[0,0,0,0],[8.999999E+09,8.999999E+09,8.999999E+09,8.999999E+09,8.999999E+09,8.999999E+09]];
	LOCAL CONST Robtarget Tr_meulage_bavure_P109 :=[[35.5770859375,158.162015625,23],[0.399851735576571,-0.390910707705398,-0.579554500955597,0.592810246689257],[0,0,0,0],[8.999999E+09,8.999999E+09,8.999999E+09,8.999999E+09,8.999999E+09,8.999999E+09]];
	LOCAL CONST Robtarget Tr_meulage_bavure_P110 :=[[35.01833984375,159.51971875,23],[0.400274548150781,-0.39012823485125,-0.578761769397268,0.593813995084891],[0,0,0,0],[8.999999E+09,8.999999E+09,8.999999E+09,8.999999E+09,8.999999E+09,8.999999E+09]];
	LOCAL CONST Robtarget Tr_meulage_bavure_P111 :=[[30.874755859375,169.745,23],[0.400461528868352,-0.389116068124019,-0.578119906266483,0.594976153641941],[0,0,0,0],[8.999999E+09,8.999999E+09,8.999999E+09,8.999999E+09,8.999999E+09,8.999999E+09]];
	LOCAL CONST Robtarget Tr_meulage_bavure_P112 :=[[30.62188671875,170.37915625,23],[0.400479922365682,-0.387966298751388,-0.577594063630269,0.596224018699515],[0,0,0,0],[8.999999E+09,8.999999E+09,8.999999E+09,8.999999E+09,8.999999E+09,8.999999E+09]];
	LOCAL CONST Robtarget Tr_meulage_bavure_P113 :=[[27.69543359375,177.2771875,23],[0.400416364321847,-0.386792673464427,-0.577139749480314,0.597467884080237],[0,0,0,0],[8.999999E+09,8.999999E+09,8.999999E+09,8.999999E+09,8.999999E+09,8.999999E+09]];
	LOCAL CONST Robtarget Tr_meulage_bavure_P114 :=[[27.010375,178.90903125,23],[0.400359652643635,-0.385710595674478,-0.576713095688454,0.598616312992677],[0,0,0,0],[8.999999E+09,8.999999E+09,8.999999E+09,8.999999E+09,8.999999E+09,8.999999E+09]];
	LOCAL CONST Robtarget Tr_meulage_bavure_P115 :=[[26.92367578125,179.108484375,23],[0.400372662837898,-0.384810559492382,-0.576288908772393,0.599594577845042],[0,0,0,0],[8.999999E+09,8.999999E+09,8.999999E+09,8.999999E+09,8.999999E+09,8.999999E+09]];
	LOCAL CONST Robtarget Tr_meulage_bavure_P116 :=[[26.85284375,179.29690625,23],[0.400462041847915,-0.384124150250067,-0.575876796761006,0.60037047327958],[0,0,0,0],[8.999999E+09,8.999999E+09,8.999999E+09,8.999999E+09,8.999999E+09,8.999999E+09]];
	LOCAL CONST Robtarget Tr_meulage_bavure_P117 :=[[24.422455078125,184.97428125,23],[0.400562703216415,-0.383612864994942,-0.575531417380388,0.600961128701725],[0,0,0,0],[8.999999E+09,8.999999E+09,8.999999E+09,8.999999E+09,8.999999E+09,8.999999E+09]];
	LOCAL CONST Robtarget Tr_meulage_bavure_P118 :=[[23.460357421875,187.456390625,23],[0.400545447221073,-0.383171010384059,-0.575344747004166,0.601433074918932],[0,0,0,0],[8.999999E+09,8.999999E+09,8.999999E+09,8.999999E+09,8.999999E+09,8.999999E+09]];
	LOCAL CONST Robtarget Tr_meulage_bavure_P119 :=[[23.18994140625,188.25540625,23],[0.400207636691959,-0.382620323237794,-0.575453419747122,0.601904392308435],[0,0,0,0],[8.999999E+09,8.999999E+09,8.999999E+09,8.999999E+09,8.999999E+09,8.999999E+09]];
	LOCAL CONST Robtarget Tr_meulage_bavure_P120 :=[[21.537169921875,192.348140625,23],[0.399328682379751,-0.381758177737248,-0.576000978823304,0.602511551386513],[0,0,0,0],[8.999999E+09,8.999999E+09,8.999999E+09,8.999999E+09,8.999999E+09,8.999999E+09]];
	LOCAL CONST Robtarget Tr_meulage_bavure_P121 :=[[20.54113671875,194.856015625,23],[0.397687573907908,-0.380368815934734,-0.577123544745518,0.603400838186373],[0,0,0,0],[8.999999E+09,8.999999E+09,8.999999E+09,8.999999E+09,8.999999E+09,8.999999E+09]];
	LOCAL CONST Robtarget Tr_meulage_bavure_P122 :=[[20.41030859375,195.169375,23],[0.394907403303714,-0.378083091760567,-0.579049442816735,0.604816551786008],[0,0,0,0],[8.999999E+09,8.999999E+09,8.999999E+09,8.999999E+09,8.999999E+09,8.999999E+09]];
	LOCAL CONST Robtarget Tr_meulage_bavure_P123 :=[[19.064513671875,197.7046875,23],[0.39040382855383,-0.37432070262587,-0.582118581329724,0.607129985675931],[0,0,0,0],[8.999999E+09,8.999999E+09,8.999999E+09,8.999999E+09,8.999999E+09,8.999999E+09]];
	LOCAL CONST Robtarget Tr_meulage_bavure_P124 :=[[18.2406015625,199.65628125,23],[0.3831039896948,-0.368010482982638,-0.586925531908365,0.610997575681684],[0,0,0,0],[8.999999E+09,8.999999E+09,8.999999E+09,8.999999E+09,8.999999E+09,8.999999E+09]];
	LOCAL CONST Robtarget Tr_meulage_bavure_P125 :=[[17.452087890625,201.56153125,23],[0.371190835602684,-0.357355669066191,-0.594401949602798,0.617414456956774],[0,0,0,0],[8.999999E+09,8.999999E+09,8.999999E+09,8.999999E+09,8.999999E+09,8.999999E+09]];
	LOCAL CONST Robtarget Tr_meulage_bavure_P126 :=[[16.77941796875,203.42984375,23],[0.352059107367655,-0.339774887862426,-0.605642303724765,0.627538692382012],[0,0,0,0],[8.999999E+09,8.999999E+09,8.999999E+09,8.999999E+09,8.999999E+09,8.999999E+09]];
	LOCAL CONST Robtarget Tr_meulage_bavure_P127 :=[[16.368560546875,204.297453125,23],[0.322551545638851,-0.312111589815149,-0.62140260993713,0.642188175126553],[0,0,0,0],[8.999999E+09,8.999999E+09,8.999999E+09,8.999999E+09,8.999999E+09,8.999999E+09]];
	LOCAL CONST Robtarget Tr_meulage_bavure_P128 :=[[14.878234375,208.698734375,23],[0.280091212983151,-0.271746609924291,-0.64112070600172,0.660807788044404],[0,0,0,0],[8.999999E+09,8.999999E+09,8.999999E+09,8.999999E+09,8.999999E+09,8.999999E+09]];
	LOCAL CONST Robtarget Tr_meulage_bavure_P129 :=[[13.8171083984375,211.01828125,23],[0.224948833902961,-0.218812352450899,-0.662038863062508,0.680605407218826],[0,0,0,0],[8.999999E+09,8.999999E+09,8.999999E+09,8.999999E+09,8.999999E+09,8.999999E+09]];
	LOCAL CONST Robtarget Tr_meulage_bavure_P130 :=[[10.760314453125,214.431765625,23],[0.162601621365722,-0.158550502574803,-0.679889266920621,0.697261095708528],[0,0,0,0],[8.999999E+09,8.999999E+09,8.999999E+09,8.999999E+09,8.999999E+09,8.999999E+09]];
	LOCAL CONST Robtarget Tr_meulage_bavure_P131 :=[[10.7413330078125,214.450015625,23],[0.101911093137242,-0.099588814475668,-0.691779326958378,0.707910700526498],[0,0,0,0],[8.999999E+09,8.999999E+09,8.999999E+09,8.999999E+09,8.999999E+09,8.999999E+09]];
	LOCAL CONST Robtarget Tr_meulage_bavure_P132 :=[[10.7346494140625,214.456,23],[0.0491899894511892,-0.0481576278343657,-0.697909117828305,0.712870290495596],[0,0,0,0],[8.999999E+09,8.999999E+09,8.999999E+09,8.999999E+09,8.999999E+09,8.999999E+09]];
	LOCAL CONST Robtarget Tr_meulage_bavure_P133 :=[[10.732666015625,214.46740625,23],[0.00518272129894051,-0.00508128323196718,-0.700065891128709,0.714041362974738],[0,0,0,0],[8.999999E+09,8.999999E+09,8.999999E+09,8.999999E+09,8.999999E+09,8.999999E+09]];
	LOCAL CONST Robtarget Tr_meulage_bavure_P134 :=[[10.29425,214.457390625,23],[0.0330276107991734,-0.0324139296145542,0.699694657524713,-0.712941722950211],[0,0,0,0],[8.999999E+09,8.999999E+09,8.999999E+09,8.999999E+09,8.999999E+09,8.999999E+09]];
	LOCAL CONST Robtarget Tr_meulage_bavure_P135 :=[[7.36895751953125,214.369265625,23],[0.0689225593649623,-0.0676796150098717,0.697367345382716,-0.71017458143513],[0,0,0,0],[8.999999E+09,8.999999E+09,8.999999E+09,8.999999E+09,8.999999E+09,8.999999E+09]];
	LOCAL CONST Robtarget Tr_meulage_bavure_P136 :=[[7.2083740234375,214.316953125,23],[0.104402212716218,-0.102530821988756,0.693141190223411,-0.705792390818958],[0,0,0,0],[8.999999E+09,8.999999E+09,8.999999E+09,8.999999E+09,8.999999E+09,8.999999E+09]];
	LOCAL CONST Robtarget Tr_meulage_bavure_P137 :=[[5.14642333984375,213.547125,23],[0.139062759878285,-0.136524894236616,0.687133764692478,-0.69990691630263],[0,0,0,0],[8.999999E+09,8.999999E+09,8.999999E+09,8.999999E+09,8.999999E+09,8.999999E+09]];
	LOCAL CONST Robtarget Tr_meulage_bavure_P138 :=[[3.53399658203125,212.337578125,23],[0.170802436203504,-0.167565075219064,0.679967082413452,-0.693104061586653],[0,0,0,0],[8.999999E+09,8.999999E+09,8.999999E+09,8.999999E+09,8.999999E+09,8.999999E+09]];
	LOCAL CONST Robtarget Tr_meulage_bavure_P139 :=[[2.55044555664063,211.6225625,23],[0.197377834100193,-0.193434089191734,0.672676090346123,-0.686390647678956],[0,0,0,0],[8.999999E+09,8.999999E+09,8.999999E+09,8.999999E+09,8.999999E+09,8.999999E+09]];
	LOCAL CONST Robtarget Tr_meulage_bavure_P140 :=[[1.69430541992188,210.9166875,23],[0.217639822158674,-0.213012374138047,0.666244519357734,-0.680717912721999],[0,0,0,0],[8.999999E+09,8.999999E+09,8.999999E+09,8.999999E+09,8.999999E+09,8.999999E+09]];
	LOCAL CONST Robtarget Tr_meulage_bavure_P141 :=[[-0.01507568359375,209.505734375,23],[0.231686956798619,-0.226424845330373,0.661246385525096,-0.676613745867247],[0,0,0,0],[8.999999E+09,8.999999E+09,8.999999E+09,8.999999E+09,8.999999E+09,8.999999E+09]];
	LOCAL CONST Robtarget Tr_meulage_bavure_P142 :=[[-3.91754150390625,205.94890625,23],[0.240549231669157,-0.234714071299472,0.657748746038113,-0.674100852219232],[0,0,0,0],[8.999999E+09,8.999999E+09,8.999999E+09,8.999999E+09,8.999999E+09,8.999999E+09]];
	LOCAL CONST Robtarget Tr_meulage_bavure_P143 :=[[-4.7983095703125,205.187140625,23],[0.245578367463917,-0.239240984874714,0.655510752989653,-0.67287492842643],[0,0,0,0],[8.999999E+09,8.999999E+09,8.999999E+09,8.999999E+09,8.999999E+09,8.999999E+09]];
	LOCAL CONST Robtarget Tr_meulage_bavure_P144 :=[[-5.47747802734375,204.60840625,23],[0.248044257320818,-0.241282179838577,0.654191404738049,-0.672525510348393],[0,0,0,0],[8.999999E+09,8.999999E+09,8.999999E+09,8.999999E+09,8.999999E+09,8.999999E+09]];
	LOCAL CONST Robtarget Tr_meulage_bavure_P145 :=[[-11.9626162109375,199.055390625,23],[0.248936712842317,-0.241825036284658,0.653477311227656,-0.672695004096105],[0,0,0,0],[8.999999E+09,8.999999E+09,8.999999E+09,8.999999E+09,8.999999E+09,8.999999E+09]];
	LOCAL CONST Robtarget Tr_meulage_bavure_P146 :=[[-12.5148623046875,198.589328125,23],[0.248941856661178,-0.241563510020946,0.653152460992384,-0.673102433013013],[0,0,0,0],[8.999999E+09,8.999999E+09,8.999999E+09,8.999999E+09,8.999999E+09,8.999999E+09]];
	LOCAL CONST Robtarget Tr_meulage_bavure_P147 :=[[-16.366759765625,195.2628125,23],[0.248552406099965,-0.240989773543681,0.653053778127728,-0.673547617724526],[0,0,0,0],[8.999999E+09,8.999999E+09,8.999999E+09,8.999999E+09,8.999999E+09,8.999999E+09]];
	LOCAL CONST Robtarget Tr_meulage_bavure_P148 :=[[-18.384796875,193.597328125,23],[0.248035305186601,-0.240374859426783,0.653099787522193,-0.673913259904426],[0,0,0,0],[8.999999E+09,8.999999E+09,8.999999E+09,8.999999E+09,8.999999E+09,8.999999E+09]];
	LOCAL CONST Robtarget Tr_meulage_bavure_P149 :=[[-21.129974609375,191.301484375,23],[0.247517757896062,-0.239851317634695,0.653257208842874,-0.674137466730507],[0,0,0,0],[8.999999E+09,8.999999E+09,8.999999E+09,8.999999E+09,8.999999E+09,8.999999E+09]];
	LOCAL CONST Robtarget Tr_meulage_bavure_P150 :=[[-22.790130859375,189.801296875,23],[0.24699199468099,-0.239408268388897,0.653525773199362,-0.674227483387255],[0,0,0,0],[8.999999E+09,8.999999E+09,8.999999E+09,8.999999E+09,8.999999E+09,8.999999E+09]];
	LOCAL CONST Robtarget Tr_meulage_bavure_P151 :=[[-28.993896484375,184.83725,23],[0.246288197182167,-0.238884134940625,0.653970364815657,-0.674239761468651],[0,0,0,0],[8.999999E+09,8.999999E+09,8.999999E+09,8.999999E+09,8.999999E+09,8.999999E+09]];
	LOCAL CONST Robtarget Tr_meulage_bavure_P152 :=[[-31.529357421875,182.671390625,23],[0.245193893401591,-0.238068228997137,0.654661589699474,-0.674256387402369],[0,0,0,0],[8.999999E+09,8.999999E+09,8.999999E+09,8.999999E+09,8.999999E+09,8.999999E+09]];
	LOCAL CONST Robtarget Tr_meulage_bavure_P153 :=[[-37.65283203125,177.354796875,23],[0.243576452106119,-0.236817615129339,0.655630110505298,-0.674341966173438],[0,0,0,0],[8.999999E+09,8.999999E+09,8.999999E+09,8.999999E+09,8.999999E+09,8.999999E+09]];
	LOCAL CONST Robtarget Tr_meulage_bavure_P154 :=[[-41.10827734375,174.4675,23],[0.241472900843959,-0.235160063521929,0.656854181984731,-0.674487335901524],[0,0,0,0],[8.999999E+09,8.999999E+09,8.999999E+09,8.999999E+09,8.999999E+09,8.999999E+09]];
	LOCAL CONST Robtarget Tr_meulage_bavure_P155 :=[[-42.819703125,173.0050625,23],[0.239131187895687,-0.23331868092725,0.658225909301122,-0.674623836245561],[0,0,0,0],[8.999999E+09,8.999999E+09,8.999999E+09,8.999999E+09,8.999999E+09,8.999999E+09]];
	LOCAL CONST Robtarget Tr_meulage_bavure_P156 :=[[-48.39929296875,168.44684375,23],[0.236927541582488,-0.231642969660352,0.659594494386309,-0.67464211076828],[0,0,0,0],[8.999999E+09,8.999999E+09,8.999999E+09,8.999999E+09,8.999999E+09,8.999999E+09]];
	LOCAL CONST Robtarget Tr_meulage_bavure_P157 :=[[-49.81979296875,167.277765625,23],[0.235219580523282,-0.23046977936001,0.660821637279594,-0.674440652276623],[0,0,0,0],[8.999999E+09,8.999999E+09,8.999999E+09,8.999999E+09,8.999999E+09,8.999999E+09]];
	LOCAL CONST Robtarget Tr_meulage_bavure_P158 :=[[-57.07016015625,161.34346875,23],[0.234223068296645,-0.22999983534865,0.661818255888052,-0.673970493560806],[0,0,0,0],[8.999999E+09,8.999999E+09,8.999999E+09,8.999999E+09,8.999999E+09,8.999999E+09]];
	LOCAL CONST Robtarget Tr_meulage_bavure_P159 :=[[-68.8285234375,151.64071875,23],[0.233965775472933,-0.230250910942493,0.662557615606964,-0.673247309626051],[0,0,0,0],[8.999999E+09,8.999999E+09,8.999999E+09,8.999999E+09,8.999999E+09,8.999999E+09]];
	LOCAL CONST Robtarget Tr_meulage_bavure_P160 :=[[-69.378390625,151.199890625,23],[0.234345142886645,-0.231108035715043,0.663049522539239,-0.672336790971504],[0,0,0,0],[8.999999E+09,8.999999E+09,8.999999E+09,8.999999E+09,8.999999E+09,8.999999E+09]];
	LOCAL CONST Robtarget Tr_meulage_bavure_P161 :=[[-69.82696875,150.84384375,23],[0.235202743902523,-0.232408277708893,0.6633329158596,-0.671308799622284],[0,0,0,0],[8.999999E+09,8.999999E+09,8.999999E+09,8.999999E+09,8.999999E+09,8.999999E+09]];
	LOCAL CONST Robtarget Tr_meulage_bavure_P162 :=[[-70.2732265625,150.48575,23],[0.23637654906504,-0.233985802667499,0.663451580462324,-0.670230386944813],[0,0,0,0],[8.999999E+09,8.999999E+09,8.999999E+09,8.999999E+09,8.999999E+09,8.999999E+09]];
	LOCAL CONST Robtarget Tr_meulage_bavure_P163 :=[[-73.0738203125,148.227390625,23],[0.237713010465013,-0.235679125200126,0.663444814807281,-0.669170271534755],[0,0,0,0],[8.999999E+09,8.999999E+09,8.999999E+09,8.999999E+09,8.999999E+09,8.999999E+09]];
	LOCAL CONST Robtarget Tr_meulage_bavure_P164 :=[[-76.844453125,145.248171875,23],[0.239041231264227,-0.237313576698826,0.663366784695941,-0.66819612766931],[0,0,0,0],[8.999999E+09,8.999999E+09,8.999999E+09,8.999999E+09,8.999999E+09,8.999999E+09]];
	LOCAL CONST Robtarget Tr_meulage_bavure_P165 :=[[-78.5739765625,143.8109375,23],[0.240177446549751,-0.238699781528676,0.663277285250752,-0.6673832866782],[0,0,0,0],[8.999999E+09,8.999999E+09,8.999999E+09,8.999999E+09,8.999999E+09,8.999999E+09]];
	LOCAL CONST Robtarget Tr_meulage_bavure_P166 :=[[-81.6443515625,141.229921875,23],[0.240955927139954,-0.239675948617189,0.663243803111787,-0.66678582653232],[0,0,0,0],[8.999999E+09,8.999999E+09,8.999999E+09,8.999999E+09,8.999999E+09,8.999999E+09]];
	LOCAL CONST Robtarget Tr_meulage_bavure_P167 :=[[-87.12621875,136.537625,23],[0.241319354109392,-0.24018118083795,0.663286671649606,-0.666429861962608],[0,0,0,0],[8.999999E+09,8.999999E+09,8.999999E+09,8.999999E+09,8.999999E+09,8.999999E+09]];
	LOCAL CONST Robtarget Tr_meulage_bavure_P168 :=[[-91.408234375,132.9519375,23],[0.241347265714954,-0.240297455520254,0.663383378734881,-0.666281564371024],[0,0,0,0],[8.999999E+09,8.999999E+09,8.999999E+09,8.999999E+09,8.999999E+09,8.999999E+09]];
	LOCAL CONST Robtarget Tr_meulage_bavure_P169 :=[[-94.813046875,130.10934375,23],[0.241225323172235,-0.240220163617278,0.663480585199457,-0.666256804479718],[0,0,0,0],[8.999999E+09,8.999999E+09,8.999999E+09,8.999999E+09,8.999999E+09,8.999999E+09]];
	LOCAL CONST Robtarget Tr_meulage_bavure_P170 :=[[-101.1326328125,124.852109375,23],[0.241186205307115,-0.240178713679279,0.663491676931705,-0.66627486408184],[0,0,0,0],[8.999999E+09,8.999999E+09,8.999999E+09,8.999999E+09,8.999999E+09,8.999999E+09]];
	LOCAL CONST Robtarget Tr_meulage_bavure_P171 :=[[-104.15115625,122.41784375,23],[0.241382809398814,-0.24033544210295,0.663373690634455,-0.666264632987477],[0,0,0,0],[8.999999E+09,8.999999E+09,8.999999E+09,8.999999E+09,8.999999E+09,8.999999E+09]];
	LOCAL CONST Robtarget Tr_meulage_bavure_P172 :=[[-111.2348359375,116.55615625,23],[0.241822831664314,-0.240704235585015,0.66313141957901,-0.666213111117167],[0,0,0,0],[8.999999E+09,8.999999E+09,8.999999E+09,8.999999E+09,8.999999E+09,8.999999E+09]];
	LOCAL CONST Robtarget Tr_meulage_bavure_P173 :=[[-111.9009375,116.001796875,23],[0.242376551675933,-0.241157339981928,0.66281346752023,-0.666164433037619],[0,0,0,0],[8.999999E+09,8.999999E+09,8.999999E+09,8.999999E+09,8.999999E+09,8.999999E+09]];
	LOCAL CONST Robtarget Tr_meulage_bavure_P174 :=[[-115.810671875,112.58215625,23],[0.242847980127083,-0.24150653696693,0.662499106179481,-0.666178944024671],[0,0,0,0],[8.999999E+09,8.999999E+09,8.999999E+09,8.999999E+09,8.999999E+09,8.999999E+09]];
	LOCAL CONST Robtarget Tr_meulage_bavure_P175 :=[[-116.085421875,112.345640625,23],[0.243074294781255,-0.241590549850314,0.662248179665958,-0.666315422280427],[0,0,0,0],[8.999999E+09,8.999999E+09,8.999999E+09,8.999999E+09,8.999999E+09,8.999999E+09]];
	LOCAL CONST Robtarget Tr_meulage_bavure_P176 :=[[-116.25915625,112.201234375,23],[0.242987499393448,-0.241341034247645,0.662083880267762,-0.666600716933593],[0,0,0,0],[8.999999E+09,8.999999E+09,8.999999E+09,8.999999E+09,8.999999E+09,8.999999E+09]];
	LOCAL CONST Robtarget Tr_meulage_bavure_P177 :=[[-122.39065625,107.259671875,23],[0.242620028384791,-0.240790915940921,0.661993977293882,-0.667022661274355],[0,0,0,0],[8.999999E+09,8.999999E+09,8.999999E+09,8.999999E+09,8.999999E+09,8.999999E+09]];
	LOCAL CONST Robtarget Tr_meulage_bavure_P178 :=[[-126.3987734375,103.733,23],[0.242070540559658,-0.240037695218397,0.661940635738475,-0.667546517499371],[0,0,0,0],[8.999999E+09,8.999999E+09,8.999999E+09,8.999999E+09,8.999999E+09,8.999999E+09]];
	LOCAL CONST Robtarget Tr_meulage_bavure_P179 :=[[-127.969296875,102.4123828125,23],[0.241457733275511,-0.239202531066965,0.661883953880808,-0.668124197861234],[0,0,0,0],[8.999999E+09,8.999999E+09,8.999999E+09,8.999999E+09,8.999999E+09,8.999999E+09]];
	LOCAL CONST Robtarget Tr_meulage_bavure_P180 :=[[-128.9561171875,101.5568515625,23],[0.240898786582222,-0.23838945554499,0.661766631519425,-0.668732508194128],[0,0,0,0],[8.999999E+09,8.999999E+09,8.999999E+09,8.999999E+09,8.999999E+09,8.999999E+09]];
	LOCAL CONST Robtarget Tr_meulage_bavure_P181 :=[[-130.3146953125,100.430359375,23],[0.240485235884319,-0.237692165602696,0.661559943042852,-0.669333793778488],[0,0,0,0],[8.999999E+09,8.999999E+09,8.999999E+09,8.999999E+09,8.999999E+09,8.999999E+09]];
	LOCAL CONST Robtarget Tr_meulage_bavure_P182 :=[[-133.451140625,97.876859375,23],[0.240281450888164,-0.237174774342021,0.66124252471129,-0.669903929148299],[0,0,0,0],[8.999999E+09,8.999999E+09,8.999999E+09,8.999999E+09,8.999999E+09,8.999999E+09]];
	LOCAL CONST Robtarget Tr_meulage_bavure_P183 :=[[-135.980625,95.83728125,23],[0.240313882565643,-0.236860053182966,0.660802240664505,-0.670437880631128],[0,0,0,0],[8.999999E+09,8.999999E+09,8.999999E+09,8.999999E+09,8.999999E+09,8.999999E+09]];
	LOCAL CONST Robtarget Tr_meulage_bavure_P184 :=[[-142.561546875,90.380984375,23],[0.240561482562188,-0.236733605445804,0.660255842565322,-0.670931885900849],[0,0,0,0],[8.999999E+09,8.999999E+09,8.999999E+09,8.999999E+09,8.999999E+09,8.999999E+09]];
	LOCAL CONST Robtarget Tr_meulage_bavure_P185 :=[[-144.058140625,89.1706875,23],[0.240983528121517,-0.236758750622937,0.659623203732026,-0.671393671608446],[0,0,0,0],[8.999999E+09,8.999999E+09,8.999999E+09,8.999999E+09,8.999999E+09,8.999999E+09]];
	LOCAL CONST Robtarget Tr_meulage_bavure_P186 :=[[-146.326,87.2804296875,23],[0.241538002012742,-0.236899181800668,0.658926332849214,-0.671829040101538],[0,0,0,0],[8.999999E+09,8.999999E+09,8.999999E+09,8.999999E+09,8.999999E+09,8.999999E+09]];
	LOCAL CONST Robtarget Tr_meulage_bavure_P187 :=[[-152.09625,82.3843046875,23],[0.24220059395985,-0.237138734601974,0.658184110127845,-0.672233419291311],[0,0,0,0],[8.999999E+09,8.999999E+09,8.999999E+09,8.999999E+09,8.999999E+09,8.999999E+09]];
	LOCAL CONST Robtarget Tr_meulage_bavure_P188 :=[[-152.93071875,81.7033984375,23],[0.242964020375825,-0.237484499460739,0.657417359276124,-0.672586063668514],[0,0,0,0],[8.999999E+09,8.999999E+09,8.999999E+09,8.999999E+09,8.999999E+09,8.999999E+09]];
	LOCAL CONST Robtarget Tr_meulage_bavure_P189 :=[[-157.892375,77.578734375,23],[0.243811166039999,-0.237941499971817,0.656659476817636,-0.672858298166089],[0,0,0,0],[8.999999E+09,8.999999E+09,8.999999E+09,8.999999E+09,8.999999E+09,8.999999E+09]];
	LOCAL CONST Robtarget Tr_meulage_bavure_P190 :=[[-163.65771875,72.8828125,23],[0.24470738136893,-0.238489358360443,0.655939360517527,-0.673041364832981],[0,0,0,0],[8.999999E+09,8.999999E+09,8.999999E+09,8.999999E+09,8.999999E+09,8.999999E+09]];
	LOCAL CONST Robtarget Tr_meulage_bavure_P191 :=[[-164.68784375,72.0086953125,23],[0.245593168667271,-0.239083576100678,0.655294341413934,-0.673136215972487],[0,0,0,0],[8.999999E+09,8.999999E+09,8.999999E+09,8.999999E+09,8.999999E+09,8.999999E+09]];
	LOCAL CONST Robtarget Tr_meulage_bavure_P192 :=[[-165.313609375,71.42959375,23],[0.246389441638743,-0.23967144084053,0.654781585516903,-0.673135141529799],[0,0,0,0],[8.999999E+09,8.999999E+09,8.999999E+09,8.999999E+09,8.999999E+09,8.999999E+09]];
	LOCAL CONST Robtarget Tr_meulage_bavure_P193 :=[[-168.852921875,68.3090546875,23],[0.247030691255316,-0.240207797984896,0.654446154284555,-0.673035127246212],[0,0,0,0],[8.999999E+09,8.999999E+09,8.999999E+09,8.999999E+09,8.999999E+09,8.999999E+09]];
	LOCAL CONST Robtarget Tr_meulage_bavure_P194 :=[[-170.8588125,66.595640625,23],[0.247463822485032,-0.240662367570033,0.654332121363324,-0.672824461764624],[0,0,0,0],[8.999999E+09,8.999999E+09,8.999999E+09,8.999999E+09,8.999999E+09,8.999999E+09]];
	LOCAL CONST Robtarget Tr_meulage_bavure_P195 :=[[-179.64409375,59.10723828125,23],[0.247636156131749,-0.241003206462414,0.654481191430296,-0.672493984147894],[0,0,0,0],[8.999999E+09,8.999999E+09,8.999999E+09,8.999999E+09,8.999999E+09,8.999999E+09]];
	LOCAL CONST Robtarget Tr_meulage_bavure_P196 :=[[-181.469078125,57.591828125,23],[0.247502174277774,-0.241196925477245,0.654922958859867,-0.672043625686856],[0,0,0,0],[8.999999E+09,8.999999E+09,8.999999E+09,8.999999E+09,8.999999E+09,8.999999E+09]];
	LOCAL CONST Robtarget Tr_meulage_bavure_P197 :=[[-185.09575,54.65811328125,23],[0.24702993993577,-0.241228370077693,0.655689238529229,-0.671458639621198],[0,0,0,0],[8.999999E+09,8.999999E+09,8.999999E+09,8.999999E+09,8.999999E+09,8.999999E+09]];
	LOCAL CONST Robtarget Tr_meulage_bavure_P198 :=[[-193.064109375,47.86023046875,23],[0.246215474173142,-0.241106716686304,0.656799343003743,-0.67071612063249],[0,0,0,0],[8.999999E+09,8.999999E+09,8.999999E+09,8.999999E+09,8.999999E+09,8.999999E+09]];
	LOCAL CONST Robtarget Tr_meulage_bavure_P199 :=[[-195.1120625,46.04815625,23],[0.245111568698056,-0.240891163607872,0.658246298761541,-0.669778751792528],[0,0,0,0],[8.999999E+09,8.999999E+09,8.999999E+09,8.999999E+09,8.999999E+09,8.999999E+09]];
	LOCAL CONST Robtarget Tr_meulage_bavure_P200 :=[[-204.501125,38.68667578125,23],[0.243820460923481,-0.240685096785728,0.659999764844882,-0.668597470399797],[0,0,0,0],[8.999999E+09,8.999999E+09,8.999999E+09,8.999999E+09,8.999999E+09,8.999999E+09]];
	LOCAL CONST Robtarget Tr_meulage_bavure_P201 :=[[-207.28975,36.442140625,23],[0.242460316104383,-0.240606000914093,0.662019768628416,-0.667121857971892],[0,0,0,0],[8.999999E+09,8.999999E+09,8.999999E+09,8.999999E+09,8.999999E+09,8.999999E+09]];
	LOCAL CONST Robtarget Tr_meulage_bavure_P202 :=[[-213.825640625,30.845671875,23],[0.241168549055643,-0.240792847975967,0.664258443367408,-0.665294863744735],[0,0,0,0],[8.999999E+09,8.999999E+09,8.999999E+09,8.999999E+09,8.999999E+09,8.999999E+09]];
	LOCAL CONST Robtarget Tr_meulage_bavure_P203 :=[[-217.468546875,27.72155859375,23],[0.24023097984849,-0.241530174480825,0.666603267377731,-0.663017597849129],[0,0,0,0],[8.999999E+09,8.999999E+09,8.999999E+09,8.999999E+09,8.999999E+09,8.999999E+09]];
	LOCAL CONST Robtarget Tr_meulage_bavure_P204 :=[[-221.793625,24.062408203125,23],[0.240138997668858,-0.243317979535269,0.668858429178556,-0.660119704561427],[0,0,0,0],[8.999999E+09,8.999999E+09,8.999999E+09,8.999999E+09,8.999999E+09,8.999999E+09]];
	LOCAL CONST Robtarget Tr_meulage_bavure_P205 :=[[-228.361390625,18.533203125,23],[0.241712463686258,-0.247003209225219,0.670681713758952,-0.656315883062811],[0,0,0,0],[8.999999E+09,8.999999E+09,8.999999E+09,8.999999E+09,8.999999E+09,8.999999E+09]];
	LOCAL CONST Robtarget Tr_meulage_bavure_P206 :=[[-229.451625,17.614533203125,23],[0.246169223188598,-0.253871638726818,0.6715274449704,-0.651153434496363],[0,0,0,0],[8.999999E+09,8.999999E+09,8.999999E+09,8.999999E+09,8.999999E+09,8.999999E+09]];
